PROGRAM MainState
VAR
	iMainSetp :INT;
	I1: UINT;
	iErrorSetp: INT;
	iLightSel: INT;
	bTurnOn: BOOL;
	bDoor_Stop: BOOL;
	I2: INT;
	I4: INT;
	I5: INT;
	i: UINT;
	iCode2: ICode;
	ExtSetVel: LREAL;
	ExtSetPos: LREAL;
	ExtSetAcc: LREAL;
	ExtSetDec: DINT;
	InitSetp: INT;
	rtStoping: R_TRIG;
	iMainInitSetp: INT;
	iMainEStopSetp: INT;
	K1: UINT;
	bInitReset: BOOL;
	DA1: INT;
	Code1: BOOL;
	Code2: BOOL;
	Code3: BOOL;
	Code4: BOOL;
	CyCtrl: INT;
	bWaterOn: BOOL;
	
	Execute: BOOL;
	bCoeWrite_GlueFeed: BOOL;
	bWaterOn2: BOOL;
	arrError:					ARRAY[1..10]OF BOOL;
	bEncloserEstop:BOOL;//外罩急停汇总
	bBoxEstop:BOOL;//按钮盒急停汇总
	F: INT;
	D195: MS_Alarm;
	D196: MS_Alarm;
	D197: MS_Alarm;
	D198: MS_Alarm;
	D199: MS_Alarm;
	D200: MS_Alarm;
	D201: MS_Alarm;
	D202: MS_Alarm;
	D203: MS_Alarm;
	D204: MS_Alarm;
	D205: MS_Alarm;
	D206: MS_Alarm;
	AnFD1: MS_Alarm;
	AnFD2: MS_Alarm;
	AnFD3: MS_Alarm;
	CaFD1: MS_Alarm;
	CaFD2: MS_Alarm;
	CaFD3: MS_Alarm;
	K2:INT;
	tCycleTimer: TON;
	bSave: BOOL;
	testii2: INT;
	bReadDataFirstCyle: BOOL;
	bReadDataCyle2: BOOL;
	bSaveTest: BOOL;
	rtSaveData: R_TRIG;
	CleanTrig: R_TRIG;
	CaCibang: R_TRIG;
	AnCibang: R_TRIG;
	CaCleanBrush:R_TRIG;
	AnCleanBrush:R_TRIG;
	
END_VAR

VAR
	R_TRIG_Bt: 			ARRAY[1..10]OF R_TRIG;
	TON20:Tc2_Standard.TON;	
//	TON21:Tc2_Standard.TON;	
	rt100:Tc2_Standard.R_TRIG;
	rt101:Tc2_Standard.R_TRIG;

	tDelayBuzze:TON;
	FanTon:TON;//除尘风机计时
	FanTonS:REAL;//除尘风机寿命秒
	FanTonH:REAL;//除尘风机寿命小时
	FanTonH_Set:REAL;//除尘风机寿命设定小时
	aAirAlarm_TON:TON;//气压报警延时；
	aTime:ARRAY[1..99] OF TON;//延时备用，1-16风速仪报警延时；
	aAlarm:ARRAY[1..99] OF BOOL;//报警预留;   1、气压不足报警；2、正极R角清废料报警；3、负极R角清废料报警；4、正极R角清废料计数错误；5、负极R角清废料计数错误；6、风机未启用报警；7、风机故障报警； 16-19、安全光栅报警；20-29、风速仪报警；30-47毛刷旋转感应报警，48毛刷旋转感应报警汇总,50:模切通道安全门报警；
	RT200:ARRAY[1..4] OF Tc2_Standard.R_TRIG;
	K3:INT;
	K4:INT;
	
	csAxis                 :ARRAY[1..MaxAxes] OF   CS_AxisCtrl;
	fbCy                   :ARRAY[1..MaxCy]    OF   FB_CylinderV2;
    fbRec                 :ARRAY[1..MaxRec]   OF   FB_Rectify;
	fbDustMotor       :ARRAY[1..MaxDust]   OF   CS_DustMoter;


    csCodeTcp:CS_CodeTcp;
    fbCamInTest: MC_CamIn;//主轴与驱动凸轮耦合

//速度模式验证
	MC_ExtSetPointGenDisable: MC_ExtSetPointGenDisable;
	MC_ExtSetPointGenEnable: MC_ExtSetPointGenEnable;
    MC_ExtSetPointGenOut:        Tc2_MC2.ST_McOutputs;
    MC_ExtSetPointGenOut2:        Tc2_MC2.ST_McOutputs;

    tonEStop:                     Tc2_Standard.TON;
   
  fbAnSetp1Moter  : CS_SetpMoter;
  fbCaSetp1Moter:CS_SetpMoter;
 // fbP4CutElectric_CY   :FB_Electric_CY;   电缸


	mc_Home    :MC_Home;

     fbCoeWrite_GlueFeed:       FB_EcCoeSdoWrite;
     	wEncodeHome                    :WORD:=6;
	test:ARRAY[1..10] OF BOOL;
	bAnReady:BOOL;//正极准备好
	bCaReady:BOOL;//负极准备好
	//fbDataXML       : FB_DataXML;
	rt10:Tc2_Standard.R_TRIG;
	testii:INT:=0;
	
	Code_MES				:ARRAY[1..20]OF  R_TRIG;
	fCode_MES				:ARRAY[1..20]OF  F_TRIG;
	tCode_MES				:ARRAY[1..20]OF  TON;
	
//模切直线电机COE寻址修改参数
	FB_EcCoESdoWrite_AnSEPTATCache : ARRAY[1..4] OF FB_EcCoESdoWrite; //正极极片缓存参数修改
	FB_EcCoESdoWrite_AnDriverDDR : ARRAY[1..4] OF FB_EcCoESdoWrite;	  //正极主驱参数修改
	FB_EcCoESdoWrite_CaSEPTATCache : ARRAY[1..4] OF FB_EcCoESdoWrite; //正极极片缓存参数修改
	FB_EcCoESdoWrite_CaDriverDDR : ARRAY[1..4] OF FB_EcCoESdoWrite;	  //正极主驱参数修改
	
	wSaveCoeCode  :DWORD:=16#65766173;    //电机参数保存
	
	SEPTATCache_fSmoothValue   :ARRAY[1..4] OF REAL;    //隔膜缓存写入参数值
	SEPTATCache_bWriteCoeValue  :ARRAY[1..4] OF BOOL;    //隔膜缓存写入执行	
	SEPTATCache_SavePara  :ARRAY[1..4] OF BOOL;   //隔膜缓存参数保存
	
	DriverDDR_fSmoothValue   :ARRAY[1..4] OF REAL;    //主驱写入参数值
	DriverDDR_bWriteCoeValue  :ARRAY[1..4] OF BOOL;    //主驱写入执行	
	DriverDDR_SavePara  :ARRAY[1..4] OF BOOL;   //主驱参数保存
	
	ExcelRate_R	:R_TRIG;	//Mes读取优报表	xfp20240316
	MTDWtStep: UINT;
	rDoorAlm :ARRAY[1..2]OF R_TRIG;
END_VAR

	aAirAlarm_TON(IN:=NOT I205[5],PT:=T#1S,Q=>);											
R_TRIG_Bt[1](CLK:= stSysState.btnStart OR stSysState.hmiStart);//启动上升沿
R_TRIG_Bt[2](CLK:= stSysState.btnStop  OR  stSysState.hmiStop);//停止上升沿
R_TRIG_Bt[4](CLK:=  stSysState.btnAuto OR  stSysState.hmiAuto);//手自动切换上升沿
R_TRIG_Bt[5](CLK:=  NOT stSysState.btnAuto);
R_TRIG_Bt[6](CLK:=stSysState.btnEstop);
R_TRIG_Bt[7](CLK:=stSysState.btnReset OR  stSysState.hmiReset );
R_TRIG_Bt[8](CLK:=  NOT stSysState.hmiAuto);



IF R_TRIG_Bt[4].Q THEN  //自动
	stSysState.FlgAuto:=TRUE;
	stSysState.FlgManua:=FALSE;
END_IF
IF R_TRIG_Bt[5].Q  OR  R_TRIG_Bt[8].Q   THEN  //手动
	stSysState.FlgAuto:=FALSE;
	stSysState.FlgManua:=TRUE;
	stSysState.bwindow:=FALSE;
END_IF
stSysState.bReset:=R_TRIG_Bt[7].Q  OR  bInitReset    ;  //复位

stSysState.bAnccdstate:= NOT AnAlarm.arrFlowAlarm[8] AND NOT AnAlarm.arrFlowAlarm[14] AND  ((NOT ProductPar.iModeEN.bCcdTcpEN AND NOT ProductPar.iModeEN.bSizeCCDEN  AND 
                         NOT  ProductPar.iModeEN.bChamferCCDEN AND NOT  ProductPar.iModeEN.bCuterCCDEN(* AND NOT  ProductPar.iModeEN.bLineScanCCDEN*)) OR  ProductPar.iModeEN.bP2PartEN);
stSysState.bCaccdstate:= NOT CaAlarm.arrFlowAlarm[8] AND NOT CaAlarm.arrFlowAlarm[14] AND  ((NOT ProductPar.iModeEN.bCcdTcpEN AND NOT ProductPar.iModeEN.bSizeCCDEN  AND 
                         NOT  ProductPar.iModeEN.bChamferCCDEN AND NOT  ProductPar.iModeEN.bCuterCCDEN (*AND NOT  ProductPar.iModeEN.bLineScanCCDEN*)) OR  ProductPar.iModeEN.bP2PartEN);

//////////////////////////////////系统流程///////////////////////
CASE iMainSetp OF 
0://   INIT
    Init();
    stSysState.iMode:=0;
 IF  stSysState.bInitDone THEN
     iMainSetp:=88;	
  END_IF
88://切换手动
  IF  stSysState.FlgManua THEN
	  iMainSetp:=300;
  END_IF
   
 (***********************手动*********************************) 
300:
   stSysState.iMode:=3;
   iMainSetp:=350;  
   
350: 
  	IF  R_TRIG_Bt[1].Q  AND stSysState.FlgAuto THEN  //启动按钮  
		IF stSysState.bAutoCondition THEN
		  stSysState.bwindow:=TRUE;	
	      iMainSetp:=90;
	    END_IF
	END_IF 
	
	IF  stSysState.FlgManua AND TON20.Q THEN  //系统清除
	   iMainSetp:=999;
	END_IF

 90:	
  	IF  R_TRIG_Bt[1].Q  AND stSysState.FlgAuto AND NOT stSysState.bwindow  THEN  //启动按钮  
		IF stSysState.bAutoCondition AND (stSysState.bAnccdstate OR ProductPar.iModeEN.iModeRun=1) AND (stSysState.bCaccdstate OR ProductPar.iModeEN.iModeRun=2) THEN
	      iMainSetp:=100;
	    END_IF
		
	ELSIF stSysState.FlgManua OR  stSysState.btnStop  OR  stSysState.hmiStop   OR   stSysState.bErrorStop OR 
          stSysState.btnEstop OR NOT stSysState.bAnccdstate OR NOT stSysState.bCaccdstate  THEN
		  iMainSetp:=300;
	END_IF 	
	
 (************************自动********************************) 
100:
   stSysState.iMode:=1;
   iMainSetp:=150;  
150:  //系统停止中......
    rtStoping(Clk:=stSysState.FlgManua OR  stSysState.btnStop  OR  stSysState.hmiStop   OR   stSysState.bErrorStop OR stSysState.btnEstop);  //自动中触发手动 停止 按钮  stSysRun.bErrorStop 包括正极和负极
    IF stSysState.FlgManua OR  stSysState.btnStop  OR  stSysState.hmiStop   OR   stSysState.bErrorStop OR stSysState.btnEstop THEN //自动触发停止 rtStoping.Q
		stSysState.Stoping:=TRUE;
		iMainSetp:=160; //
	END_IF;
	
160: //判断停止完成
   	IF  stSysState.bStopFinished  THEN
		AnSys.bStopFinished:=FALSE; 
		CaSys.bStopFinished:=FALSE;
       	stSysState.Stoping:=FALSE;
		IF NOT  stSysState.btnEstop THEN
			iMainSetp:=300; 
		ELSE
			stSysState.bInitDone:=FALSE;
			iMainSetp:=400; 	
		END_IF
	END_IF;
	
 (************************急停********************************) 
400://Stoping
   stSysState.iMode:=4;
    EStop();  
   iMainSetp:=450; 
      
450: //急停跳出 
	IF  NOT  stSysState.btnEstop  THEN  
        tonEStop(IN:=FALSE , PT:=T#50MS );
	    iMainSetp:=0;
    ELSE
         tonEStop(IN:=TRUE , PT:=T#50MS );
         IF  tonEStop.Q THEN
              tonEStop(IN:=FALSE , PT:=T#50MS );
              iMainSetp:=400;   
         END_IF
   	 END_IF

END_CASE


IF   stSysState.btnEstop   THEN  //AND  stSysState.iMode=3
	  iMainSetp:=400;
END_IF



(***************程序调用*********************)



AnPart(iMode:=stSysState.iMode);
CaPart(iMode:=stSysState.iMode);
//	XML();
   Condition();
    MotionBasic();
    CyBasic();
    RecBasic();
     Alarm();
     Pusle();
	 MS_Alarm();
	 Motion_coe();
	 MesCollect();
//PoleData.AnBeltData[1].Meney.SizeResults;

ACTION Alarm:

IF NOT ProductPar.iModeEN.bDoorEN THEN
	IF NOT I206[15] THEN
		aAlarm[49]:=TRUE;//模切通道安全门报警
	END_IF
END_IF



IF R_TRIG_Bt[7].Q THEN
	FOR K1:=1 TO MaxAxes DO 
     arrAxisAlarm[K1]:=  FALSE ;
END_FOR
END_IF
(******************气缸报警*******************)
FOR K1:=1 TO MaxCy DO 
     arrCYOnAlarm[K1]:=  arrCyCtrl[K1] .Status.Error1;
     arrCYOFFAlarm[K1]:=  arrCyCtrl[K1] .Status.Error2;
END_FOR
(******************正极气缸报警*******************)
bAnCYHaveAlarm:=FALSE;
FOR K1:=1 TO 20 DO 
      bAnCYHaveAlarm:=(bAnCYHaveAlarm OR arrCYOnAlarm[K1] OR  arrCYOFFAlarm[K1]) ;
END_FOR
FOR K1:=41 TO 60 DO 
      bAnCYHaveAlarm:=(bAnCYHaveAlarm OR arrCYOnAlarm[K1] OR  arrCYOFFAlarm[K1]) ;
END_FOR
(******************负极气缸报警*******************)
bCaCYHaveAlarm:=FALSE;
FOR K1:=21 TO 40 DO 
      bCaCYHaveAlarm:=(bCaCYHaveAlarm OR arrCYOnAlarm[K1] OR  arrCYOFFAlarm[K1]) ;
END_FOR
FOR K1:=61 TO MaxCy DO 
      bCaCYHaveAlarm:=(bCaCYHaveAlarm OR arrCYOnAlarm[K1] OR  arrCYOFFAlarm[K1]) ;
END_FOR

(******************切刀计数报警*************)
IF ProductPar.AnPar.iMouldCount1>= ProductPar.AnPar.iMouldCountAlarm1 THEN   //正极前模具切刀计数报警
	CuterCountAlarm[1]:=TRUE;
	ELSE
	CuterCountAlarm[1]:=FALSE;	
END_IF
(*IF ProductPar.AnPar.iMouldCount2>= ProductPar.AnPar.iMouldCountAlarm2 THEN   //正极后模具切刀计数报警
	CuterCountAlarm[2]:=TRUE;
	ELSE
	CuterCountAlarm[2]:=FALSE;	
END_IF*)
IF ProductPar.AnPar.iCuterCount>= ProductPar.AnPar.iCuterCountAlarm THEN   //正极裁切切刀计数报警
	CuterCountAlarm[3]:=TRUE;
	ELSE
	CuterCountAlarm[3]:=FALSE;	
END_IF
IF ProductPar.CaPar.iMouldCount1>= ProductPar.CaPar.iMouldCountAlarm1 THEN   //负极前模具切刀计数报警
	CuterCountAlarm[4]:=TRUE;
	ELSE
	CuterCountAlarm[4]:=FALSE;	
END_IF
(*IF ProductPar.CaPar.iMouldCount2>= ProductPar.CaPar.iMouldCountAlarm2 THEN   //负极后模具切刀计数报警
	CuterCountAlarm[5]:=TRUE;
	ELSE
	CuterCountAlarm[5]:=FALSE;	
END_IF*)
IF ProductPar.CaPar.iCuterCount>= ProductPar.CaPar.iCuterCountAlarm THEN   //负极裁切切刀计数报警
	CuterCountAlarm[6]:=TRUE;
	ELSE
	CuterCountAlarm[6]:=FALSE;	
END_IF

IF CuterCountAlarm[1] OR CuterCountAlarm[3] OR CuterCountAlarm[4] OR CuterCountAlarm[6] THEN// OR CuterCountAlarm[2] OR CuterCountAlarm[5]
	b_lifetime:=TRUE;
	ELSE
	b_lifetime:=FALSE;	
END_IF

IF ProductPar.AnPar.iCuterCount>= ProductPar.AnPar.iCuterCountWarning THEN    //正极裁切切刀计数预警
	CuterCountAlarm[7]:=TRUE;
	ELSE
	CuterCountAlarm[7]:=FALSE;	
END_IF
IF ProductPar.CaPar.iCuterCount>= ProductPar.CaPar.iCuterCountWarning THEN   //负极裁切切刀计数预警
	CuterCountAlarm[8]:=TRUE;
	ELSE
	CuterCountAlarm[8]:=FALSE;	
END_IF

(****************轴报警**************)
(*
FOR K1:=1 TO MaxAxes DO 
     arrAxisAlarm[K1]:=  arrAxis[K1] .Status.Error AND  arrAxis[K1] .Status.ErrorID<>16#42A0 OR NOT arrAxisCtrl[K1] .Status.Enabled ;
END_FOR
*)
(****************正极轴报警**************)
bAnAxisHaveAlarm:=FALSE;
FOR K1:=1 TO 15 DO 
		IF K1<>3 AND K1<>4 THEN
				arrAxisAlarm[K1]:=  arrAxis[K1] .Status.Error AND  arrAxis[K1] .Status.ErrorID<>16#42A0  ;//OR NOT arrAxisCtrl[K1] .Status.Enabled
				bAnAxisHaveAlarm:=bAnAxisHaveAlarm OR arrAxisAlarm[K1]  ;//OR arrAxisCtrl[K1] .Status.ErrorLimitSwitch
		END_IF
END_FOR

FOR K1:=18 TO 22 DO 
	  arrAxisAlarm[K1]:=  arrAxis[K1] .Status.Error AND  arrAxis[K1] .Status.ErrorID<>16#42A0  ;//OR NOT arrAxisCtrl[K1] .Status.Enabled
      bAnAxisHaveAlarm:=bAnAxisHaveAlarm OR arrAxisAlarm[K1]  ;//OR arrAxisCtrl[K1] .Status.ErrorLimitSwitch
END_FOR

FOR K1:=50 TO 52 DO 
	  arrAxisAlarm[K1]:=  arrAxis[K1] .Status.Error AND  arrAxis[K1] .Status.ErrorID<>16#42A0  ;//OR NOT arrAxisCtrl[K1] .Status.Enabled
      bAnAxisHaveAlarm:=bAnAxisHaveAlarm OR arrAxisAlarm[K1]  ;//OR arrAxisCtrl[K1] .Status.ErrorLimitSwitch
END_FOR

(****************负极轴报警**************)
bCaAxisHaveAlarm:=FALSE;
FOR K1:=25 TO 39 DO 
		IF K1<>27 AND K1<>28 THEN
				arrAxisAlarm[K1]:=  arrAxis[K1] .Status.Error AND  arrAxis[K1] .Status.ErrorID<>16#42A0  ;//OR NOT arrAxisCtrl[K1] .Status.Enabled
				bCaAxisHaveAlarm:=bCaAxisHaveAlarm OR arrAxisAlarm[K1]  ;//OR arrAxisCtrl[K1] .Status.ErrorLimitSwitch
		END_IF
END_FOR

FOR K1:=42 TO 46 DO 
	  arrAxisAlarm[K1]:=  arrAxis[K1] .Status.Error AND  arrAxis[K1] .Status.ErrorID<>16#42A0  ;//OR NOT arrAxisCtrl[K1] .Status.Enabled
      bCaAxisHaveAlarm:=bCaAxisHaveAlarm OR arrAxisAlarm[K1]  ;//OR arrAxisCtrl[K1] .Status.ErrorLimitSwitch
END_FOR

FOR K1:=56 TO 58 DO
	  arrAxisAlarm[K1]:=  arrAxis[K1] .Status.Error AND  arrAxis[K1] .Status.ErrorID<>16#42A0  ; //OR NOT arrAxisCtrl[K1] .Status.Enabled
      bCaAxisHaveAlarm:=bCaAxisHaveAlarm OR arrAxisAlarm[K1]  ;//OR arrAxisCtrl[K1] .Status.ErrorLimitSwitch
END_FOR

(******************张力报警*******************)
bAnTenHaveAlarm :=FALSE;
bCaTenHaveAlarm :=FALSE;
FOR K1:=1 TO 15 DO 
      bAnTenHaveAlarm:=bAnTenHaveAlarm OR AnAlarm.arrTenAlarm[K1];
	  bCaTenHaveAlarm:=bCaTenHaveAlarm OR CaAlarm.arrTenAlarm[K1];
END_FOR

(******************凸轮报警*******************)
bAnCreatTableHaveAlarm :=FALSE;
bCaCreatTableHaveAlarm :=FALSE;
bAnCamHaveAlarm :=FALSE;
bCaCamHaveAlarm :=FALSE;
FOR K1:=1 TO 30 DO 
      bAnCreatTableHaveAlarm:=bAnCreatTableHaveAlarm OR AnAlarm.arrCreatTableAlarm[K1];
	  bCaCreatTableHaveAlarm:=bCaCreatTableHaveAlarm OR CaAlarm.arrCreatTableAlarm[K1];
	  bAnCamHaveAlarm:=bAnCamHaveAlarm OR AnAlarm.arrCamInAlarm[K1];
	  bCaCamHaveAlarm:=bAnCamHaveAlarm OR CaAlarm.arrCamInAlarm[K1];
END_FOR

(******************齿轮报警*******************)
bAnGearHaveAlarm :=FALSE;
bCaGearHaveAlarm :=FALSE;
FOR K1:=1 TO 25 DO 
      bAnGearHaveAlarm:=bAnGearHaveAlarm OR AnAlarm.arrGearAlarm[K1];
	  bCaGearHaveAlarm:=bCaGearHaveAlarm OR CaAlarm.arrGearAlarm[K1];
END_FOR

(******************流程报警*******************)
bAnFlowHaveAlarm :=FALSE;
bCaFlowHaveAlarm :=FALSE;
FOR K1:=1 TO 50 DO 
      bAnFlowHaveAlarm:=bAnFlowHaveAlarm OR AnAlarm.arrFlowAlarm[K1];
	  bCaFlowHaveAlarm:=bCaFlowHaveAlarm OR CaAlarm.arrFlowAlarm[K1];
END_FOR

(******************提示*******************)
bAnHaveLightWarn :=FALSE;
bCaHaveLightWarn :=FALSE;
FOR K1:=1 TO 50 DO 
      bAnHaveLightWarn:=bAnHaveLightWarn OR AnAlarm.arrLightWarn[K1];
	  bCaHaveLightWarn:=bCaHaveLightWarn OR CaAlarm.arrLightWarn[K1];
END_FOR
(***DDR负数报警***)
(***DDR负数报警***)
IF arrAxisCtrl[NameNo.CaAxisNo.DriverDDR].Status.fActPos<-1 THEN
	CaAlarm.arrFlowAlarm[30]:=TRUE;
END_IF
IF arrAxisCtrl[NameNo.AnAxisNo.DriverDDR].Status.fActPos<-1 THEN
	AnAlarm.arrFlowAlarm[30]:=TRUE;
END_IF

 IF   stSysState.bReset AND  AnAlarm.arrFlowAlarm[30] THEN
	    arrAxisCtrl[NameNo.AnAxisNo.DriverDDR].Cmd.fSetPos:=360;
		arrAxisCtrl[NameNo.AnAxisNo.DriverDDR].Cmd.bSetPos:=TRUE;
		AnAlarm.arrFlowAlarm[30]:=FALSE;
ELSIF  stSysState.bReset AND CaAlarm.arrFlowAlarm[30] THEN
	    arrAxisCtrl[NameNo.CaAxisNo.DriverDDR].Cmd.fSetPos:=360;
		arrAxisCtrl[NameNo.CaAxisNo.DriverDDR].Cmd.bSetPos:=TRUE;
		CaAlarm.arrFlowAlarm[30]:=FALSE;
 END_IF

 (******************报警复位*****************)
 FOR K3:=1 TO 98 DO 
	IF   stSysState.bReset AND  aAlarm[K3]AND NOT aAlarm[52] AND NOT aAlarm[53] AND NOT aAlarm[54]  THEN
			aAlarm[K3]:=FALSE;
	END_IF
END_FOR

(***气压不足报警***)
IF aAirAlarm_TON.Q THEN
	aAlarm[1]:=TRUE;
END_IF
YL_Q[1]:=aAlarm[1];//气压报警传给叠台；
(*
(*** R角废料清洁提示***)
IF  YL_GVL2[1]>=YL_GVL2[2] THEN//正极R角清废料报警；
	aAlarm[2]:=TRUE;
END_IF

IF  YL_GVL2[1]< 0 THEN//正极R角清废料计数错误；
	aAlarm[4]:=TRUE;
END_IF
///////////////////////////
IF    YL_GVL2[3] >=YL_GVL2[4] THEN//负极R角清废料报警；
	aAlarm[3]:=TRUE;
END_IF

IF  YL_GVL2[3] < 0 THEN//负极R角清废料计数错误；
	aAlarm[5]:=TRUE;
END_IF
/////////////////////////////
//复位
IF   stSysState.bReset AND  (aAlarm[2] OR  aAlarm[4] )THEN
		YL_GVL2[1]:=0;
		aAlarm[2]:=FALSE;
		aAlarm[4]:=FALSE;
END_IF

IF   stSysState.bReset AND  (aAlarm[3] OR  aAlarm[5] )THEN
		YL_GVL2[3]:=0;
		aAlarm[3]:=FALSE;
		aAlarm[5]:=FALSE;
END_IF
*)
(*** 除尘风机报警提示***)
aAlarm[6];//风机未启用报警；
IF NOT ProductPar.iModeEN.bFounctionClose[2] THEN
		IF NOT YL_I[1] OR NOT YL_I[3] OR NOT YL_I[5] OR NOT YL_I[7] THEN//2个5.5KW的吸片风机,2个除尘风机；
			aAlarm[6]:=TRUE;//风机未启用报警；
		END_IF
		IF  YL_I[2] OR YL_I[4] OR YL_I[6] OR YL_I[8]  THEN
			aAlarm[7]:=TRUE;// 风机故障报警；
		END_IF
END_IF
FanTon(IN:=NOT aAlarm[6]AND NOT FanTon.Q,PT:=T#1S,Q=>);
IF FanTon.Q THEN
	FanTonS:=FanTonS+1;
END_IF
IF FanTonS>=3600 THEN
	FanTonH:=FanTonH+1;
	FanTonS:=0;
END_IF
IF FanTonH_Set>=FanTonH THEN
	aAlarm[61]:=TRUE;;//风机寿命报警
END_IF



(*** 除尘毛刷气缸没有升起报警***)

IF stSysState.iMode=1 AND NOT 	arrCyCtrl[NameNo.AnCYNo.PoleBrushDustPush_U].Io.DIOFFSwitch THEN
				aAlarm[8]:=TRUE;//	正极上表面毛刷除尘升降气缸位置异常；
END_IF
IF stSysState.iMode=1 AND NOT	arrCyCtrl[NameNo.AnCYNo.PoleWindDustPush_U].Io.DIOFFSwitch THEN
				aAlarm[9]:=TRUE;//	正极上表面风刀除尘升降气缸位置异常;
END_IF
IF stSysState.iMode=1 AND NOT	arrCyCtrl[NameNo.AnCYNo.PoleBrushDustPush_D].Io.DIOFFSwitch THEN
				aAlarm[10]:=TRUE;//	正极下表面毛刷除尘升降气缸位置异常;
END_IF
IF stSysState.iMode=1 AND NOT	arrCyCtrl[NameNo.AnCYNo.PoleWindDustPush_D].Io.DIOFFSwitch THEN
				aAlarm[11]:=TRUE;//	//	正极下表面风刀除尘升降气缸位置异常;
END_IF
////////////////////////
IF stSysState.iMode=1 AND NOT 	arrCyCtrl[NameNo.CaCYNo.PoleBrushDustPush_U].Io.DIOFFSwitch THEN
				aAlarm[12]:=TRUE;//	负极上表面毛刷除尘升降气缸位置异常；
END_IF
IF stSysState.iMode=1 AND NOT	arrCyCtrl[NameNo.CaCYNo.PoleWindDustPush_U].Io.DIOFFSwitch THEN
				aAlarm[13]:=TRUE;//	负极上表面风刀除尘升降气缸位置异常;
END_IF
IF stSysState.iMode=1 AND NOT	arrCyCtrl[NameNo.CaCYNo.PoleBrushDustPush_D].Io.DIOFFSwitch THEN
				aAlarm[14]:=TRUE;//	负极下表面毛刷除尘升降气缸位置异常;
END_IF
IF stSysState.iMode=1 AND NOT	arrCyCtrl[NameNo.CaCYNo.PoleWindDustPush_D].Io.DIOFFSwitch THEN
				aAlarm[15]:=TRUE;//	负极下表面风刀除尘升降气缸位置异常;
END_IF

(*** 安全光栅报警***)
IF NOT AnSenser.biSafetyCurtain_M THEN
	aAlarm[16]:=TRUE;
END_IF
IF NOT AnSenser.biSafetyCurtain_C THEN
	aAlarm[17]:=TRUE;
END_IF		
	
IF NOT CaSenser.biSafetyCurtain_M THEN
	aAlarm[18]:=TRUE;
END_IF
IF NOT CaSenser.biSafetyCurtain_C THEN
	aAlarm[19]:=TRUE;
END_IF	
	
(***************风速仪报警**************)
(***************风速仪报警**************)

aTime[1](IN:=I107[8],PT:=T#20S,Q=>	);
aTime[2](IN:=I107[9],PT:=T#20S,Q=>	);
aTime[3](IN:=I107[10],PT:=T#20S,Q=>	);
aTime[4](IN:=I107[11],PT:=T#20S,Q=>	);
aTime[5](IN:=I107[12],PT:=T#20S,Q=>	);

aTime[6](IN:=I207[8],PT:=T#20S,Q=>	);
aTime[7](IN:=I207[9],PT:=T#20S,Q=>	);
aTime[8](IN:=I207[10],PT:=T#20S,Q=>	);
aTime[9](IN:=I207[11],PT:=T#20S,Q=>	);
aTime[10](IN:=I207[12],PT:=T#20S,Q=>);

IF NOT ProductPar.iModeEN.bFounctionClose[1] THEN//风速仪屏蔽
	IF aTime[1].Q THEN
		aAlarm[20]:=TRUE;
	END_IF
	IF aTime[2].Q THEN
		aAlarm[21]:=TRUE;
	END_IF
	IF aTime[3].Q THEN
		aAlarm[22]:=TRUE;
	END_IF
	IF aTime[4].Q THEN
		aAlarm[23]:=TRUE;
	END_IF
	IF aTime[5].Q THEN
		aAlarm[24]:=TRUE;
	END_IF
	IF aTime[6].Q THEN
		aAlarm[25]:=TRUE;
	END_IF
	IF aTime[7].Q THEN
		aAlarm[26]:=TRUE;
	END_IF
	IF aTime[8].Q THEN
		aAlarm[27]:=TRUE;
	END_IF
	IF aTime[9].Q THEN
		aAlarm[28]:=TRUE;
	END_IF
	IF aTime[10].Q THEN
		aAlarm[29]:=TRUE;
	END_IF
ELSE
	FOR i:=20 TO 29 DO
		aAlarm[i]:=FALSE;
	END_FOR	
END_IF
(******************毛刷感应报警********************)
FOR K4:=30 TO 47 DO 
     aAlarm[48]:=  aAlarm[K4];
END_FOR
(*
(***********摆杆电机扭矩值设置过小报警************)
IF iTargetTorque[1]>-20 THEN
	aAlarm[50]:=TRUE;//正极；
END_IF
IF iTargetTorque[2]>-20 THEN
	aAlarm[51]:=TRUE;//负极；
END_IF
*)
(****************模切清洁报警*********************)

CleanTrig(CLK:= (ProductPar.CleanTimeHMIHour1 = System.StTime.wHour AND ProductPar.CleanTimeHMIMin1 =System.stTime.wMinute)
OR (ProductPar.CleanTimeHMIHour2 = System.StTime.wHour AND ProductPar.CleanTimeHMIMin2 =System.stTime.wMinute)
OR (ProductPar.CleanTimeHMIHour3 = System.StTime.wHour AND ProductPar.CleanTimeHMIMin3 =System.stTime.wMinute)
OR (ProductPar.CleanTimeHMIHour4 = System.StTime.wHour AND ProductPar.CleanTimeHMIMin4 =System.stTime.wMinute));
IF CleanTrig.Q THEN
	aAlarm[52]:=TRUE;//请清洁机台
END_IF
(****************磁棒校验时间报警******************)
AnCibang(CLK:= (ProductPar.CibangTimeHMIHour1 = System.StTime.wHour AND ProductPar.CibangTimeHMIDay1 =System.stTime.wDay));
CaCibang(CLK:= (ProductPar.CibangTimeHMIHour2 = System.StTime.wHour AND ProductPar.CibangTimeHMIDay2 =System.stTime.wDay));
IF AnCibang.Q THEN
	aAlarm[53]:=TRUE;//正极磁棒校验时间报警
END_IF
IF CaCibang.Q THEN
	aAlarm[54]:=TRUE;//负极磁棒校验时间报警
END_IF
(****************模切毛刷清洁时间****************)
AnCleanBrush(CLK:= (ProductPar.BrushTimeHMIHour1 = System.StTime.wHour AND ProductPar.BrushTimeHMIDay1 =System.stTime.wDay));
CaCleanBrush(CLK:= (ProductPar.BrushTimeHMIHour2 = System.StTime.wHour AND ProductPar.BrushTimeHMIDay2 =System.stTime.wDay));
IF AnCleanBrush.Q THEN
	aAlarm[62]:=TRUE;//正极毛刷清洁时间报警
END_IF
IF CaCleanBrush.Q THEN
	aAlarm[63]:=TRUE;//负极毛刷清洁时间报警
END_IF

IF NOT  DTM_Mes1.bFuncEN[0] AND NOT ProductPar.iModeEN.bP2PartEN AND (DTM_Mes1.bFuncEN[1] OR DTM_Mes1.bFuncEN[2] OR DTM_Mes1.bFuncEN[3] OR
	        DTM_Mes1.bFuncEN[4] OR DTM_Mes1.bFuncEN[5] OR DTM_Mes1.bFuncEN[6] OR DTM_Mes1.bFuncEN[7] )  THEN
		 aAlarm[64]:=TRUE;//模切有功能屏蔽报警
END_IF		
			


 AnAlarm.arrFlowAlarm[9];
AnAlarm.arrFlowAlarm[10];
AnAlarm.arrFlowAlarm[11];
AnAlarm.arrFlowAlarm[12];
AnAlarm.arrFlowAlarm[13];
CaAlarm.arrFlowAlarm[9];
CaAlarm.arrFlowAlarm[10];
CaAlarm.arrFlowAlarm[11];
CaAlarm.arrFlowAlarm[12];
CaAlarm.arrFlowAlarm[13];
(*===============================================报警信息============================================================*)
(*****************报警汇总****************)////根据实际情况汇总
//正极报警汇总
arrError[1]:=bAnAxisHaveAlarm OR bAnCYHaveAlarm OR bAnTenHaveAlarm OR bAnCreatTableHaveAlarm OR bAnCamHaveAlarm OR bAnGearHaveAlarm OR bAnFlowHaveAlarm OR aAlarm[16] OR aAlarm[17] OR aAlarm[49]
		OR AnAlarm.arrFlowAlarm[9] OR AnAlarm.arrFlowAlarm[10] OR AnAlarm.arrFlowAlarm[11] OR AnAlarm.arrFlowAlarm[12] OR AnAlarm.arrFlowAlarm[13]
		OR CaAlarm.arrFlowAlarm[9] OR CaAlarm.arrFlowAlarm[10] OR CaAlarm.arrFlowAlarm[11] OR CaAlarm.arrFlowAlarm[12] OR CaAlarm.arrFlowAlarm[13] OR CuterCountAlarm[3];
//负极报警汇总
arrError[2]:=bCaAxisHaveAlarm OR bCaCYHaveAlarm OR bCaTenHaveAlarm OR bCaCreatTableHaveAlarm OR bCaCamHaveAlarm OR bCaGearHaveAlarm OR bCaFlowHaveAlarm OR aAlarm[18] OR aAlarm[19] OR aAlarm[49]
		OR AnAlarm.arrFlowAlarm[9] OR AnAlarm.arrFlowAlarm[10] OR AnAlarm.arrFlowAlarm[11] OR AnAlarm.arrFlowAlarm[12] OR AnAlarm.arrFlowAlarm[13]
		OR CaAlarm.arrFlowAlarm[9] OR CaAlarm.arrFlowAlarm[10] OR CaAlarm.arrFlowAlarm[11] OR CaAlarm.arrFlowAlarm[12] OR CaAlarm.arrFlowAlarm[13] OR CuterCountAlarm[6];
//提示
arrError[3]:=(ProductPar.iModeEN.iModeRun=0 AND (bAnHaveLightWarn OR bCaHaveLightWarn)) OR
				   (ProductPar.iModeEN.iModeRun=1 AND bAnHaveLightWarn) OR 
				   (ProductPar.iModeEN.iModeRun=2 AND bCaHaveLightWarn);

arrError[4];
arrError[5]:=CaAlarm.arrFlowAlarm[30] OR AnAlarm.arrFlowAlarm[30] OR aAlarm[1] OR aAlarm[2] OR aAlarm[3] OR aAlarm[4] OR aAlarm[5]  OR aAlarm[6] OR aAlarm[7] OR aAlarm[8] OR aAlarm[9]
					OR aAlarm[10] OR aAlarm[11] OR aAlarm[12] OR aAlarm[13] OR aAlarm[14] OR aAlarm[15]OR aAlarm[52]OR aAlarm[53]OR aAlarm[54] ;

stSysState.bErrorStop:=(ProductPar.iModeEN.iModeRun=0 AND (arrError[1] OR arrError[2])) OR
								   (ProductPar.iModeEN.iModeRun=1 AND arrError[1]) OR 
								   (ProductPar.iModeEN.iModeRun=2 AND arrError[2])OR arrError[5] OR aAlarm[64];
								   
								   
rDoorAlm[1](CLK:=(AnAlarm.arrFlowAlarm[9] OR AnAlarm.arrFlowAlarm[10] OR AnAlarm.arrFlowAlarm[11] OR AnAlarm.arrFlowAlarm[12] OR AnAlarm.arrFlowAlarm[13]) AND NOT
                            bAnAxisHaveAlarm AND NOT bAnCYHaveAlarm AND NOT bAnTenHaveAlarm AND NOT bAnCreatTableHaveAlarm AND NOT bAnCamHaveAlarm AND NOT
                           bAnGearHaveAlarm AND NOT bAnFlowHaveAlarm AND NOT aAlarm[16] AND NOT aAlarm[17] AND NOT aAlarm[49]  AND NOT CuterCountAlarm[3] );
rDoorAlm[2](CLK:=(CaAlarm.arrFlowAlarm[9] OR CaAlarm.arrFlowAlarm[10] OR CaAlarm.arrFlowAlarm[11] OR CaAlarm.arrFlowAlarm[12] OR CaAlarm.arrFlowAlarm[13]) AND NOT 
                            bCaAxisHaveAlarm AND NOT bCaCYHaveAlarm AND NOT bCaTenHaveAlarm AND NOT bCaCreatTableHaveAlarm AND NOT bCaCamHaveAlarm AND NOT 
                            bCaGearHaveAlarm AND NOT bCaFlowHaveAlarm AND NOT aAlarm[18] AND NOT aAlarm[19] AND NOT aAlarm[49]AND NOT CuterCountAlarm[6] );
IF 	rDoorAlm[1].Q OR bCaDoorALM THEN						
	bAnDoorALM:=TRUE;
END_IF			

IF 	rDoorAlm[1].Q THEN						
	bCaDoorALM:=TRUE;
END_IF		

IF NOT stSysState.bErrorStop AND bAnDoorALM THEN
	bAnDoorALM:=FALSE;
END_IF		
	
IF NOT stSysState.bErrorStop AND bCaDoorALM THEN
	bCaDoorALM:=FALSE;
END_IF				
(*==============报警复位=========================*)
//轴  气缸报警  红灯亮       蜂鸣器 0.5秒 频率 响 8 秒后停止    

IF stSysState.iMode=3 THEN
	stSysState.bReset:=stSysState.btnReset;
END_IF

(*****蜂鸣器*****)
rt100(CLK:=stSysState.bErrorStop, Q=> );
rt101(CLK:=arrError[3]  , Q=> );
IF rt100.Q THEN
	iErrorSetp:=100;//故障报警
END_IF

IF rt101.Q THEN
	iErrorSetp:=200;//警告报警
END_IF


tDelayBuzze(IN:= , PT:= , Q=> , ET=> );
CASE iErrorSetp   OF
100:
  tDelayBuzze.PT:=T#8S;
  tDelayBuzze.IN:=TRUE;
  iErrorSetp:=500;
200:
  tDelayBuzze.PT:=T#4S;
   tDelayBuzze.IN:=TRUE;
  iErrorSetp:=600;
500:
		stSysState.boBuzzer:= Pulse._250ms.Q;  //   (NOT bError1 AND NOT bError2) AND
		IF tDelayBuzze.Q  THEN
			iErrorSetp:=0;
			tDelayBuzze.IN:=FALSE;
			stSysState.boBuzzer:=FALSE;
		END_IF
600:
	IF stSysState.iMode=1 AND NOT stSysState.bErrorStop THEN
		stSysState.boRedLight:=Pulse._1s.Q;
	END_IF
		stSysState.boBuzzer:= Pulse._1s.Q;  //    (NOT bError1 AND NOT bError2) AND
		IF tDelayBuzze.Q  THEN
			iErrorSetp:=0;
			tDelayBuzze.IN:=FALSE;
			IF stSysState.iMode=1 AND NOT stSysState.bErrorStop THEN
				stSysState.boRedLight:=FALSE;
			END_IF
			stSysState.boBuzzer:=FALSE;
		END_IF

END_CASE


(*****三色灯控制*********)
//自动   绿
    RT200[1](CLK:=stSysState.iMode=1 AND NOT stSysState.bErrorStop , Q=> ); 
   IF RT200[1].Q THEN
	  bTurnOn:=TRUE;
      iLightSel:=3;
   END_IF       
//手动  黄
    RT200[2](CLK:=stSysState.iMode=3 AND NOT stSysState.bErrorStop , Q=> ); 
   IF RT200[2].Q THEN
	  bTurnOn:=TRUE;
      iLightSel:=2;
   END_IF 

//暂停   黄
    RT200[3](CLK:=stSysState.iMode=2 AND NOT stSysState.bErrorStop , Q=> ); 
   IF RT200[3].Q THEN
	  bTurnOn:=TRUE;
      iLightSel:=2;
   END_IF 
   
//暂停   红   //急停 OR 故障
    RT200[4](CLK:=stSysState.iMode=4  OR stSysState.bErrorStop  , Q=> ); 
   IF RT200[4].Q THEN
	  bTurnOn:=TRUE;
      iLightSel:=1;
   END_IF    
   
IF bTurnOn THEN
	CASE iLightSel OF 
	  1: //红灯
		stSysState.boGreenLight:=FALSE;
		stSysState.boRedLight:=TRUE;
		stSysState.boYellowLight:=FALSE;
	
	  2://黄灯
		stSysState.boGreenLight:=FALSE;
		stSysState.boRedLight:=FALSE;
		stSysState.boYellowLight:=TRUE;
	
	  3://绿灯
		stSysState.boGreenLight:=TRUE;
		stSysState.boRedLight:=FALSE;
		stSysState.boYellowLight:=FALSE;
	
	END_CASE
   bTurnOn:=FALSE;
END_IF
arrAxis[4].Status.Homed;
arrAxis[5].Status.Homed;
arrAxis[6].Status.Homed;
arrAxis[7].Status.Homed;
arrAxis[8].Status.Homed;
arrAxis[9].Status.Homed;
arrAxis[10].Status.Homed;
arrAxis[11].Status.Homed;
arrAxis[12].Status.Homed;
arrAxis[13].Status.Homed;
arrAxis[14].Status.Homed;
arrAxis[15].Status.Homed;
arrAxis[16].Status.Homed;
arrAxis[17].Status.Homed;
arrAxis[18].Status.Homed;
arrAxis[19].Status.Homed;
arrAxis[20].Status.Homed;
arrAxis[21].Status.Homed;
arrAxis[22].Status.Homed;
arrAxis[23].Status.Homed;
arrAxis[24].Status.Homed;
arrAxis[25].Status.Homed;
arrAxis[26].Status.Homed;
arrAxis[27].Status.Homed;
arrAxis[28].Status.Homed;
arrAxis[29].Status.Homed;
arrAxis[30].Status.Homed;
arrAxis[31].Status.Homed;
arrAxis[32].Status.Homed;
arrAxis[33].Status.Homed;
arrAxis[34].Status.Homed;
arrAxis[35].Status.Homed;
arrAxis[36].Status.Homed;
arrAxis[37].Status.Homed;
arrAxis[38].Status.Homed;
arrAxis[39].Status.Homed;
arrAxis[40].Status.Homed;
arrAxis[41].Status.Homed;
arrAxis[42].Status.Homed;
arrAxis[43].Status.Homed;
arrAxis[44].Status.Homed;
arrAxis[45].Status.Homed;
arrAxis[46].Status.Homed;
arrAxis[47].Status.Homed;
arrAxis[48].Status.Homed;
arrAxis[49].Status.Homed;
arrAxis[50].Status.Homed;
arrAxis[51].Status.Homed;
arrAxis[52].Status.Homed;
arrAxis[53].Status.Homed;
arrAxis[54].Status.Homed;
arrAxis[55].Status.Homed;
arrAxis[56].Status.Homed;
arrAxis[57].Status.Homed;
arrAxis[58].Status.Homed;
arrAxis[59].Status.Homed;
arrAxis[60].Status.Homed;
END_ACTION

ACTION Condition:
//按钮汇总
stSysState.btnAuto:=AnSys.btnAuto AND CaSys.btnAuto ;
stSysState.btnStart:=AnSys.btnStart OR CaSys.btnStart;
stSysState.btnStop:=AnSys.btnStop OR CaSys.btnStop;
stSysState.btnReset:=AnSys.btnReset OR CaSys.btnReset;
bEncloserEstop:=(NOT AnBtn.EncloserEstop[1] OR NOT AnBtn.EncloserEstop[2] OR NOT AnBtn.EncloserEstop[3] OR 
						  NOT CaBtn.EncloserEstop[1] OR NOT CaBtn.EncloserEstop[2] OR NOT CaBtn.EncloserEstop[3])AND test[1] ;
bBoxEstop:=NOT AnBtn.PoleBoxEStop OR NOT AnBtn.NGBoxEStop OR  NOT CaBtn.PoleBoxEStop OR NOT CaBtn.NGBoxEStop ;

stSysState.btnEstop:=(NOT AnSys.btnEstop OR NOT CaSys.btnEstop //面板急停
								OR bEncloserEstop//外罩急停
								(*OR bBoxEstop//按钮盒急停*)
								) ;//常闭
//面板按钮灯控制
bAnReady:=AnSys.bAutoCondition1 AND AnSys.Homed AND NOT AnSys.hmiDisCamAll;
bCaReady:=CaSys.bAutoCondition1 AND CaSys.Homed AND NOT CaSys.hmiDisCamAll;

AnSys.boStartLight:=stSysState.boGreenLight OR bAnReady AND Pulse._500ms.Q OR AnSys.btnStart;
CaSys.boStartLight:=stSysState.boGreenLight OR bCaReady AND Pulse._500ms.Q OR AnSys.btnStart;

AnSys.boStopLight:=AnSys.Stoping AND Pulse._250ms.Q OR AnSys.btnStop;
CaSys.boStopLight:=CaSys.Stoping AND Pulse._250ms.Q OR CaSys.btnStop;

AnSys.boResetLight:=stSysState.boRedLight AND Pulse._500ms.Q OR AnSys.btnReset;
CaSys.boResetLight:=stSysState.boRedLight AND Pulse._500ms.Q OR CaSys.btnReset;		
////////////////////////////////////////////设备状态//////////////////////
	IF stSysState.btnEstop THEN
		stSysState.iModehmi:=4;
	ELSIF NOT stSysState.btnEstop AND stSysState.bErrorStop THEN
		stSysState.iModehmi:=5;
	ELSIF NOT stSysState.btnEstop AND NOT stSysState.bErrorStop AND stSysState.FlgManua AND stSysState.iMode=3THEN
		stSysState.iModehmi:=3;
	ELSIF NOT stSysState.btnEstop AND NOT stSysState.bErrorStop AND ((NOT stSysState.FlgManua AND stSysState.FlgAuto AND stSysState.iMode=1) OR stSysState.iMode=1) THEN
		stSysState.iModehmi:=1;
	ELSIF NOT stSysState.btnEstop AND NOT stSysState.bErrorStop AND NOT stSysState.FlgManua AND stSysState.FlgAuto AND stSysState.iMode<>1 AND
		 	((ProductPar.iModeEN.iModeRun=0 AND bAnReady AND bCaReady) OR (ProductPar.iModeEN.iModeRun=1 AND bAnReady) OR (ProductPar.iModeEN.iModeRun=2 AND bCaReady))
			THEN	
		stSysState.iModehmi:=2;	
	ELSE
		stSysState.iModehmi:=6;	
	END_IF		
	P2Interaction.bP1Runing:=stSysState.iModehmi=1;
////////////////////////////////////////////主流程与分模块交互//////////////////////
(*
stSysState.bAutoCondition:=((AnSys.bAutoCondition1 AND AnSys.Homed AND NOT AnSys.hmiDisCamAll AND 
			CaSys.bAutoCondition1 AND CaSys.Homed AND NOT CaSys.hmiDisCamAll AND
			ProductPar.iModeEN.iModeRun=0) OR//正负同时启用
			(AnSys.bAutoCondition1 AND AnSys.Homed AND NOT AnSys.hmiDisCamAll AND
			ProductPar.iModeEN.iModeRun=1) OR//仅正极启用
			(CaSys.bAutoCondition1 AND CaSys.Homed AND NOT CaSys.hmiDisCamAll AND
			ProductPar.iModeEN.iModeRun=2))//仅负极启用
			AND NOT stSysState.bErrorStop;
*)
stSysState.bAutoCondition:=	(AnSys.bAutoCondition1 AND AnSys.Homed AND NOT AnSys.hmiDisCamAll AND CaSys.bAutoCondition1 AND CaSys.Homed AND NOT CaSys.hmiDisCamAll AND ProductPar.iModeEN.iModeRun=0 
	AND	( (ProductPar.AnPar.MQ.bWindSelect AND  Ansys.PolePieceNumberOK1)  OR ( NOT ProductPar.AnPar.MQ.bWindSelect AND  Ansys.PolePieceNumberOK2) )
	AND  ( ( ProductPar.CaPar.MQ.bWindSelect AND  Casys.PolePieceNumberOK1 ) OR (  NOT ProductPar.CaPar.MQ.bWindSelect AND  Casys.PolePieceNumberOK2 ) ) ) OR //正负同时启用

		(AnSys.bAutoCondition1 AND AnSys.Homed AND NOT AnSys.hmiDisCamAll AND ProductPar.iModeEN.iModeRun=1  AND
		 ( ( ProductPar.AnPar.MQ.bWindSelect AND  Ansys.PolePieceNumberOK1 ) OR (  NOT ProductPar.AnPar.MQ.bWindSelect AND  Ansys.PolePieceNumberOK2 ) )) OR//仅正极启用
	
		(CaSys.bAutoCondition1 AND CaSys.Homed AND NOT CaSys.hmiDisCamAll AND ProductPar.iModeEN.iModeRun=2 AND 
		  ( ( ProductPar.CaPar.MQ.bWindSelect AND  Casys.PolePieceNumberOK1 ) OR (  NOT ProductPar.CaPar.MQ.bWindSelect AND  Casys.PolePieceNumberOK2 )  ) )//仅负极启用
		  AND NOT stSysState.bErrorStop; 			
Ansys.bAutoTen:=stSysState.iMode=1 AND (ProductPar.iModeEN.iModeRun=0 OR ProductPar.iModeEN.iModeRun=1);
Casys.bAutoTen:=stSysState.iMode=1 AND (ProductPar.iModeEN.iModeRun=0 OR ProductPar.iModeEN.iModeRun=2);
Ansys.bAutoMain:=AnSys.bAutoCondition2 AND ((ProductPar.iModeEN.iModeRun=0 AND CaSys.bAutoCondition2) OR ProductPar.iModeEN.iModeRun=1);
Casys.bAutoMain:=CaSys.bAutoCondition2 AND ((ProductPar.iModeEN.iModeRun=0 AND AnSys.bAutoCondition2) OR ProductPar.iModeEN.iModeRun=2);

stSysState.bStopFinished:=(AnSys.bStopFinished AND CaSys.bStopFinished  AND ProductPar.iModeEN.iModeRun=0) OR//正负同时启用
			(AnSys.bStopFinished AND ProductPar.iModeEN.iModeRun=1) OR//仅正极启用
			(CaSys.bStopFinished AND ProductPar.iModeEN.iModeRun=2);//仅负极启用

///////////////////////////////////交互映射/////////////////////////////////////
//////////叠片TO模切//////////
//一号叠台正极
AnInter.M1Done:=D_Pro.bAn_M1Done;
AnInter.M1Safety:=D_Pro.bAn_M1Safety;
AnInter.iM1Ask:=D_Sys.iAn1Ask;
AnInter.M1LockReady:=D_Pro.bAn_M1LockReady;
AnInter.M1JumpReady:=D_Pro.bAn_M1JumpReady;
AnInter.M1PoleHave:=D_Pro.bAn_M1PoleHave;


//一号叠台负极
CaInter.M1Done:=D_Pro.bCa_M1Done;
CaInter.M1Safety:=D_Pro.bCa_M1Safety;
CaInter.iM1Ask:=D_Sys.iCa1Ask;
CaInter.M1LockReady:=D_Pro.bCa_M1LockReady;
CaInter.M1JumpReady:=D_Pro.bCa_M1JumpReady;
CaInter.M1PoleHave:=D_Pro.bCa_M1PoleHave;


//二号叠台正极
AnInter.M2Done:=D_Pro.bAn_M2Done;
AnInter.M2Safety:=D_Pro.bAn_M2Safety;
AnInter.iM2Ask:=D_Sys.iAn2Ask;
AnInter.M2LockReady:=D_Pro.bAn_M2LockReady;
AnInter.M2JumpReady:=D_Pro.bAn_M2JumpReady;
AnInter.M2PoleHave:=D_Pro.bAn_M2PoleHave;


//二号叠台负极
CaInter.M2Done:=D_Pro.bCa_M2Done;
CaInter.M2Safety:=D_Pro.bCa_M2Safety;
CaInter.iM2Ask:=D_Sys.iCa2Ask;
CaInter.M2LockReady:=D_Pro.bCa_M2LockReady;
CaInter.M2JumpReady:=D_Pro.bCa_M2JumpReady;
CaInter.M2PoleHave:=D_Pro.bCa_M2PoleHave;


//三号叠台正极
AnInter.M3Done:=D_Pro.bAn_M3Done;
AnInter.M3Safety:=D_Pro.bAn_M3Safety;
AnInter.iM3Ask:=D_Sys.iAn3Ask;
AnInter.M3LockReady:=D_Pro.bAn_M3LockReady;
AnInter.M3JumpReady:=D_Pro.bAn_M3JumpReady;
AnInter.M3PoleHave:=D_Pro.bAn_M3PoleHave;


//三号叠台负极
CaInter.M3Done:=D_Pro.bCa_M3Done;
CaInter.M3Safety:=D_Pro.bCa_M3Safety;
CaInter.iM3Ask:=D_Sys.iCa3Ask;
CaInter.M3LockReady:=D_Pro.bCa_M3LockReady;
CaInter.M3JumpReady:=D_Pro.bCa_M3JumpReady;
CaInter.M3PoleHave:=D_Pro.bCa_M3PoleHave;


//公共
P2Interaction.bP2ClearDo:=D_Sys.bP2ClearDo;
P2Interaction.bP2ClearDone:=D_Sys.bP2ClearDone;
P2Interaction.P2M1Enable:=D_Sys.bP2M1Enable;//叠台工位：1=屏蔽   模切工位：1=启用，故取反。
P2Interaction.P2M2Enable:=D_Sys.bP2M2Enable;//叠台工位：1=屏蔽   模切工位：1=启用，故取反。
P2Interaction.P2M3Enable:=D_Sys.bP2M3Enable;//叠台工位：1=屏蔽   模切工位：1=启用，故取反。
P2Interaction.bP2Estop:=D_Sys.bP2Estop;
P2Interaction.bP2Runing:=D_Sys.bP2Runing;
P2Interaction.bP2Start:=D_Sys.bP2Start;

///////////模切TO叠片/////////
//一号叠台正极
M_Pro.bAn_M1Allow:=AnInter.M1Allow;
M_Pro.bAn_M1Allow2:=AnInter.M1Allow2;
//一号叠台负极
M_Pro.bCa_M1Allow:=CaInter.M1Allow;
//M_Pro.bCa_M1Allow:=CaInter.M1Allow2;
//二号叠台正极
M_Pro.bAn_M2Allow:=AnInter.M2Allow;
//M_Pro.bAn_M2Allow2:=AnInter.M2Allow2;
//二号叠台负极
M_Pro.bCa_M2Allow:=CaInter.M2Allow;
//M_Pro.bCa_M2Allow:=CaInter.M2Allow2;
//三号叠台正极
M_Pro.bAn_M3Allow:=AnInter.M3Allow;
//M_Pro.bAn_M3Allow2:=AnInter.M3Allow2;
//三号叠台负极
M_Pro.bCa_M3Allow:=CaInter.M3Allow;
//M_Pro.bCa_M3Allow:=CaInter.M3Allow2;

(*20240404
///////////模切TO叠片/////////
//一号叠台正极
M_Pro.bAn_M1Allow:=AnInter.M1Allow;
//一号叠台负极
M_Pro.bCa_M1Allow:=CaInter.M1Allow;
//二号叠台正极
M_Pro.bAn_M2Allow:=AnInter.M2Allow;
//二号叠台负极
M_Pro.bCa_M2Allow:=CaInter.M2Allow;
//三号叠台正极
M_Pro.bAn_M3Allow:=AnInter.M3Allow;
//三号叠台负极
M_Pro.bCa_M3Allow:=CaInter.M3Allow;
20240404*)
//公共
M_Sys.bP1ClearDo:=P2Interaction.bP1ClearDo;
M_Sys.bP1ClearDone:=P2Interaction.bP1ClearDone;
M_Sys.bP1Estop:=P2Interaction.bP1Estop;
M_Sys.bP1Runing:=P2Interaction.bP1Runing;
M_Sys.bP1Start:=P2Interaction.bP1Start;
M_Sys.iCarryPoleMode:=ProductPar.iModeEN.iCarryPoleMode;
M_Sys.p1state:=stSysState.iModehmi;
IF test[2] THEN
	MEMSET(ADR(PoleData.AnIntervalData),0,SIZEOF(PoleData.AnIntervalData)); //  
	test[2]:=FALSE;
END_IF
IF test[3] THEN
	MEMSET(ADR(PoleData.CaIntervalData),0,SIZEOF(PoleData.CaIntervalData)); //  
	test[3]:=FALSE;
END_IF
IF test[4] THEN
	MEMSET(ADR(PoleData.AnTabData),0,SIZEOF(PoleData.AnTabData)); //  
	test[4]:=FALSE;
END_IF
IF test[5] THEN
	MEMSET(ADR(PoleData.CaTabData),0,SIZEOF(PoleData.CaTabData)); //  
	test[5]:=FALSE;
END_IF
//监控
PoleData.	AnBeltData[1].bHavePole;
PoleData.	AnBeltData[2].bHavePole;
PoleData.	AnBeltData[3].bHavePole;
PoleData.	AnBeltData[4].bHavePole;
PoleData.	AnBeltData[5].bHavePole;
PoleData.	AnBeltData[6].bHavePole;
PoleData.	AnBeltData[7].bHavePole;
PoleData.	AnBeltData[8].bHavePole;
PoleData.	AnBeltData[9].bHavePole;
PoleData.	AnBeltData[10].bHavePole;
PoleData.	AnBeltData[11].bHavePole;
PoleData.	AnBeltData[12].bHavePole;
PoleData.	AnBeltData[13].bHavePole;
PoleData.	AnBeltData[14].bHavePole;
PoleData.	AnBeltData[15].bHavePole;
PoleData.	AnBeltData[16].bHavePole;
PoleData.	AnBeltData[17].bHavePole;
PoleData.	AnBeltData[18].bHavePole;
PoleData.	AnBeltData[19].bHavePole;
PoleData.	AnBeltData[20].bHavePole;
PoleData.	AnBeltData[21].bHavePole;
PoleData.	AnBeltData[22].bHavePole;
PoleData.	AnBeltData[23].bHavePole;
PoleData.	AnBeltData[24].bHavePole;
PoleData.	AnBeltData[25].bHavePole;
PoleData.	AnBeltData[26].bHavePole;
PoleData.	AnBeltData[27].bHavePole;
PoleData.	AnBeltData[28].bHavePole;
PoleData.	AnBeltData[29].bHavePole;
PoleData.	AnBeltData[30].bHavePole;				
stSysState.hmiStart;					
bInitReset;
arrAxisCtrl[NameNo.AnVirAxisNo.VirMain].Status.fModuloActPos;
arrAxisCtrl[NameNo.AnVirAxisNo.VirDriver].Status.fActPos;
arrAxisCtrl[NameNo.AnVirAxisNo.VirBelt].Status.fActPos;
arrAxisCtrl[NameNo.AnAxisNo.Mould].Status.fModuloActPos;
arrAxisCtrl[NameNo.AnAxisNo.Cuter].Status.fModuloActPos;
arrAxisCtrl[NameNo.AnAxisNo.DriverDDR].Status.fActPos;
arrAxisCtrl[NameNo.AnAxisNo.CCDPressPush].Status.fModuloActPos;
//arrAxisCtrl[NameNo.AnAxisNo.NGPush2].Status.fModuloActPos;
arrAxisCtrl[NameNo.AnAxisNo.CuterBelt].Status.fActPos;
arrAxisCtrl[NameNo.AnAxisNo.NGPushReverseBelt].Status.fActPos;
arrAxisCtrl[NameNo.AnAxisNo.DedustBelt].Status.fActPos;
arrAxisCtrl[NameNo.AnAxisNo.DedustReverseBelt].Status.fActPos;
arrAxisCtrl[NameNo.AnAxisNo.SubBelt1].Status.fActPos;
arrAxisCtrl[NameNo.AnAxisNo.SubBelt2].Status.fActPos;
arrAxisCtrl[NameNo.AnAxisNo.SubBelt3].Status.fActPos;

arrAxisCtrl[NameNo.AnAxisNo.CuterBeltChange].Status.Homed;
arrAxisCtrl[NameNo.AnAxisNo.CuterBeltChange].cmd.bHome;

PoleData.	CaBeltData[1].bHavePole;
PoleData.	CaBeltData[2].bHavePole;
PoleData.	CaBeltData[3].bHavePole;
PoleData.	CaBeltData[4].bHavePole;
PoleData.	CaBeltData[5].bHavePole;
PoleData.	CaBeltData[6].bHavePole;
PoleData.	CaBeltData[7].bHavePole;
PoleData.	CaBeltData[8].bHavePole;
PoleData.	CaBeltData[9].bHavePole;
PoleData.	CaBeltData[10].bHavePole;
PoleData.	CaBeltData[11].bHavePole;
PoleData.	CaBeltData[12].bHavePole;
PoleData.	CaBeltData[13].bHavePole;
PoleData.	CaBeltData[14].bHavePole;
PoleData.	CaBeltData[15].bHavePole;
PoleData.	CaBeltData[16].bHavePole;
PoleData.	CaBeltData[17].bHavePole;
PoleData.	CaBeltData[18].bHavePole;
PoleData.	CaBeltData[19].bHavePole;
PoleData.	CaBeltData[20].bHavePole;
PoleData.	CaBeltData[21].bHavePole;
PoleData.	CaBeltData[22].bHavePole;
PoleData.	CaBeltData[23].bHavePole;
PoleData.	CaBeltData[24].bHavePole;
PoleData.	CaBeltData[25].bHavePole;
PoleData.	CaBeltData[26].bHavePole;
PoleData.	CaBeltData[27].bHavePole;
PoleData.	CaBeltData[28].bHavePole;
PoleData.	CaBeltData[29].bHavePole;
PoleData.	CaBeltData[30].bHavePole;	




//正极左卷料号OK
IF  (ProductPar.AnPar.MQ.bWindSelect AND arrCyCtrl[NameNo.AnCYNo.Inflation_L].Status.ONState 
 AND DT_To_MQ_MES.Mes_PcToPlc1 AND  LEN(DT_To_MQ_MES.PostiveCode1)>6  )  OR ProductPar.iModeEN.PartNumberOff THEN
	Ansys.PolePieceNumberOK1:=TRUE;
ELSE
	Ansys.PolePieceNumberOK1:=FALSE;
END_IF

//正极右卷料号OK
IF  (NOT ProductPar.AnPar.MQ.bWindSelect AND arrCyCtrl[NameNo.AnCYNo.Inflation_R].Status.ONState
  AND DT_To_MQ_MES.Mes_PcToPlc2 AND LEN(DT_To_MQ_MES.PostiveCode2)>6  )  OR ProductPar.iModeEN.PartNumberOff THEN
	Ansys.PolePieceNumberOK2:=TRUE;
ELSE
	Ansys.PolePieceNumberOK2:=FALSE;
END_IF

//当前使用左卷
IF ProductPar.AnPar.MQ.bWindSelect THEN
	IF Ansys.PolePieceNumberOK1 THEN
		PoleData.AnBeltData[1].Code:=DT_To_MQ_MES.PostiveCode1;
	ELSE
		PoleData.AnBeltData[1].Code:='';//当前卷物料码异常
	END_IF
ELSE//当前使用右卷
	IF Ansys.PolePieceNumberOK2 THEN
		PoleData.AnBeltData[1].Code:=DT_To_MQ_MES.PostiveCode2;
	ELSE
		PoleData.AnBeltData[1].Code:='';//当前卷物料码异常
	END_IF
END_IF

//正极右卷换左卷---正常换卷
Code_MES[1](CLK:=ProductPar.AnPar.MQ.bWindSelect , Q=> );//AND arrCyCtrl[NameNo.AnCYNo.Inflation_L].Status.ONState  AND  stAnUwindTen.bTensionOK 
IF Code_MES[1].Q THEN
	Ansys.PolePieceNumberOK2:=FALSE;//正极右卷料号OK
	MQ_To_DT_MES.Mes_PlcToPc1:=FALSE;//正极左卷换卷请求
	MQ_To_DT_MES.Mes_PlcToPc2:=TRUE;//正极右卷换卷请求触发
END_IF
//正极左卷换右卷---正常换卷
Code_MES[2](CLK:=NOT ProductPar.AnPar.MQ.bWindSelect  , Q=> );//AND arrCyCtrl[NameNo.AnCYNo.Inflation_R].Status.ONState  AND  stAnUwindTen.bTensionOK
IF Code_MES[2].Q THEN
	Ansys.PolePieceNumberOK1:=FALSE;//正极左卷料号OK
	MQ_To_DT_MES.Mes_PlcToPc1:=TRUE;//正极左卷换卷请求触发
	MQ_To_DT_MES.Mes_PlcToPc2:=FALSE;//正极右卷换卷请求
END_IF

//正极气涨轴切换换卷
Code_MES[3](CLK:=arrCyCtrl[NameNo.AnCYNo.Inflation_L].Io.DOStatus1, Q=> );//左卷
Code_MES[4](CLK:=arrCyCtrl[NameNo.AnCYNo.Inflation_R].Io.DOStatus1, Q=> );//右卷
IF Code_MES[3].Q THEN//左卷请求
	Ansys.PolePieceNumberOK1:=FALSE;//正极左卷料号OK
	MQ_To_DT_MES.Mes_PlcToPc1:=TRUE;//正极左卷换卷请求触发
	MQ_To_DT_MES.Mes_PlcToPc2:=FALSE;//正极右卷换卷请求
END_IF
IF Code_MES[4].Q THEN//右卷请求
	Ansys.PolePieceNumberOK2:=FALSE;//正极右卷料号OK
	MQ_To_DT_MES.Mes_PlcToPc1:=FALSE;//正极左卷换卷请求
	MQ_To_DT_MES.Mes_PlcToPc2:=TRUE;//正极右卷换卷请求触发
END_IF



//负极左卷料号OK
IF  (ProductPar.CaPar.MQ.bWindSelect AND arrCyCtrl[NameNo.CaCYNo.Inflation_L].Status.ONState 
 AND DT_To_MQ_MES.Mes_PcToPlc3 AND  LEN(DT_To_MQ_MES.NegativeCode1)>6  )  OR ProductPar.iModeEN.PartNumberOff THEN
	Casys.PolePieceNumberOK1:=TRUE;
ELSE
	Casys.PolePieceNumberOK1:=FALSE;
END_IF

//负极右卷料号OK
IF  (NOT ProductPar.CaPar.MQ.bWindSelect AND arrCyCtrl[NameNo.CaCYNo.Inflation_R].Status.ONState
  AND DT_To_MQ_MES.Mes_PcToPlc4 AND LEN(DT_To_MQ_MES.NegativeCode2)>6  )  OR ProductPar.iModeEN.PartNumberOff THEN
	Casys.PolePieceNumberOK2:=TRUE;
ELSE
	Casys.PolePieceNumberOK2:=FALSE;
END_IF

IF ProductPar.CaPar.MQ.bWindSelect THEN
	IF  Casys.PolePieceNumberOK1 THEN
		PoleData.CaBeltData[1].Code:=DT_To_MQ_MES.NegativeCode1;
	ELSE
		PoleData.CaBeltData[1].Code:='';//当前卷物料码异常
	END_IF
ELSE
	IF  Casys.PolePieceNumberOK2 THEN
		PoleData.CaBeltData[1].Code:=DT_To_MQ_MES.NegativeCode2;
	ELSE
		PoleData.CaBeltData[1].Code:='';//当前卷物料码异常
	END_IF
END_IF

//负极右卷换左卷---正常换卷
Code_MES[5](CLK:=ProductPar.CaPar.MQ.bWindSelect  , Q=> );//AND arrCyCtrl[NameNo.CaCYNo.Inflation_L].Status.ONState  AND  stCaUwindTen.bTensionOK
IF Code_MES[5].Q THEN
	Casys.PolePieceNumberOK2:=FALSE;//负极右卷料号OK
	MQ_To_DT_MES.Mes_PlcToPc3:=FALSE;//负极左卷换卷请求
	MQ_To_DT_MES.Mes_PlcToPc4:=TRUE;//负极右卷换卷请求触发
END_IF
//正极左卷换右卷---正常换卷
Code_MES[6](CLK:=NOT ProductPar.CaPar.MQ.bWindSelect  , Q=> );//AND arrCyCtrl[NameNo.CaCYNo.Inflation_R].Status.ONState  AND  stCaUwindTen.bTensionOK
IF Code_MES[6].Q THEN
	Casys.PolePieceNumberOK1:=FALSE;//负极左卷料号OK
	MQ_To_DT_MES.Mes_PlcToPc3:=TRUE;//负极左卷换卷请求触发
	MQ_To_DT_MES.Mes_PlcToPc4:=FALSE;//负极右卷换卷请求
END_IF


//负极气涨轴切换换卷
Code_MES[7](CLK:=arrCyCtrl[NameNo.CaCYNo.Inflation_L].Io.DOStatus1, Q=> );//左卷
Code_MES[8](CLK:=arrCyCtrl[NameNo.CaCYNo.Inflation_R].Io.DOStatus1, Q=> );//右卷
IF Code_MES[7].Q THEN//左卷请求
	Casys.PolePieceNumberOK1:=FALSE;//负极左卷料号OK
	MQ_To_DT_MES.Mes_PlcToPc3:=TRUE;//负极左卷换卷请求触发
	MQ_To_DT_MES.Mes_PlcToPc4:=FALSE;//负极右卷换卷请求
END_IF
IF Code_MES[8].Q THEN//右卷请求
	Casys.PolePieceNumberOK2:=FALSE;//负极右卷料号OK
	MQ_To_DT_MES.Mes_PlcToPc3:=FALSE;//负极左卷换卷请求
	MQ_To_DT_MES.Mes_PlcToPc4:=TRUE;//负极右卷换卷请求触发
END_IF



//条码校验未完成提示
IF ProductPar.AnPar.MQ.bWindSelect AND  NOT Ansys.PolePieceNumberOK1  AND NOT ProductPar.iModeEN.PartNumberOff THEN
	AnAlarm.arrLightWarn[41]:=TRUE;//正极左卷物料码校验未通过
ELSE
	AnAlarm.arrLightWarn[41]:=FALSE;//正极左卷物料码校验未通过
END_IF
IF NOT ProductPar.AnPar.MQ.bWindSelect AND NOT Ansys.PolePieceNumberOK2  AND NOT ProductPar.iModeEN.PartNumberOff THEN
	AnAlarm.arrLightWarn[42]:=TRUE;//正极右卷物料码校验未通过
ELSE
	AnAlarm.arrLightWarn[42]:=FALSE;//正极右卷物料码校验未通过
END_IF

IF ProductPar.CaPar.MQ.bWindSelect AND  NOT Casys.PolePieceNumberOK1  AND NOT ProductPar.iModeEN.PartNumberOff THEN
	CaAlarm.arrLightWarn[41]:=TRUE;//负极左卷物料码校验未通过
ELSE
	CaAlarm.arrLightWarn[41]:=FALSE;//负极左卷物料码校验未通过
END_IF
IF NOT  ProductPar.CaPar.MQ.bWindSelect AND NOT Casys.PolePieceNumberOK2  AND NOT ProductPar.iModeEN.PartNumberOff THEN
	CaAlarm.arrLightWarn[42]:=TRUE;//负极右卷物料码校验未通过
ELSE
	CaAlarm.arrLightWarn[42]:=FALSE;//负极右卷物料码校验未通过
END_IF


//触发信号清除
tCode_MES[1](IN:=MQ_To_DT_MES.Mes_PlcToPc1 , PT:=T#0.2S , Q=> , ET=> );
tCode_MES[2](IN:=MQ_To_DT_MES.Mes_PlcToPc2 , PT:=T#0.2S , Q=> , ET=> );
tCode_MES[3](IN:=MQ_To_DT_MES.Mes_PlcToPc3 , PT:=T#0.2S , Q=> , ET=> );
tCode_MES[4](IN:=MQ_To_DT_MES.Mes_PlcToPc4 , PT:=T#0.2S , Q=> , ET=> );
IF tCode_MES[1].Q THEN
	MQ_To_DT_MES.Mes_PlcToPc1:=FALSE;//正极左卷换卷请求触发
END_IF
IF tCode_MES[2].Q THEN
	MQ_To_DT_MES.Mes_PlcToPc2:=FALSE;//正极右卷换卷请求触发
END_IF
IF tCode_MES[3].Q THEN
	MQ_To_DT_MES.Mes_PlcToPc3:=FALSE;//负极左卷换卷请求触发
END_IF
IF tCode_MES[4].Q THEN
	MQ_To_DT_MES.Mes_PlcToPc4:=FALSE;//负极右卷换卷请求触发
END_IF


//料号相同检测
IF  NOT ProductPar.iModeEN.PartNumberOff  THEN
	IF DT_To_MQ_MES.PostiveCode1 =DT_To_MQ_MES.PostiveCode2 AND DT_To_MQ_MES.PostiveCode1<>''  THEN
		aAlarm[55]:=TRUE;;//正极左卷和正极右卷料号相同
	END_IF
	IF DT_To_MQ_MES.PostiveCode1 =DT_To_MQ_MES.NegativeCode1 AND DT_To_MQ_MES.PostiveCode1<>''  THEN
		aAlarm[56]:=TRUE;;//正极左卷和负极左卷料号相同
	END_IF
	IF DT_To_MQ_MES.PostiveCode1 =DT_To_MQ_MES.NegativeCode2 AND DT_To_MQ_MES.PostiveCode1<>''  THEN
		aAlarm[57]:=TRUE;;//正极左卷与负极右卷料号相同
	END_IF
	
	IF DT_To_MQ_MES.PostiveCode2 =DT_To_MQ_MES.NegativeCode1 AND DT_To_MQ_MES.PostiveCode2<>''  THEN
		aAlarm[58]:=TRUE;;//正极右卷和负极左卷料号相同
	END_IF
	IF DT_To_MQ_MES.PostiveCode2 =DT_To_MQ_MES.NegativeCode2 AND DT_To_MQ_MES.PostiveCode2<>'' THEN
		aAlarm[59]:=TRUE;;//正极右卷和负极右卷料号相同
	END_IF
	
	IF DT_To_MQ_MES.NegativeCode1= DT_To_MQ_MES.NegativeCode2 AND DT_To_MQ_MES.NegativeCode1<>'' THEN 
		aAlarm[60]:=TRUE;;//负极左卷和负极右卷料号相同
	END_IF
END_IF

IF YL_I[20] THEN//叠台一正极送片流水线安全点动条件 
		arrAxisCtrl[20].Cmd.JogN_Condition:=TRUE;
		arrAxisCtrl[20].Cmd.JogP_Condition:=TRUE;
ELSE
		arrAxisCtrl[20].Cmd.JogN_Condition:=FALSE;
		arrAxisCtrl[20].Cmd.JogP_Condition:=FALSE;	
END_IF
IF YL_I[21] THEN//叠台一负极送片流水线安全点动条件 
		arrAxisCtrl[44].Cmd.JogN_Condition:=TRUE;
		arrAxisCtrl[44].Cmd.JogP_Condition:=TRUE;
ELSE
		arrAxisCtrl[44].Cmd.JogN_Condition:=FALSE;
		arrAxisCtrl[44].Cmd.JogP_Condition:=FALSE;		
END_IF

IF YL_I[22] THEN//叠台二正极送片流水线安全点动条件 
		arrAxisCtrl[21].Cmd.JogN_Condition:=TRUE;
		arrAxisCtrl[21].Cmd.JogP_Condition:=TRUE;
ELSE
		arrAxisCtrl[21].Cmd.JogN_Condition:=FALSE;
		arrAxisCtrl[21].Cmd.JogP_Condition:=FALSE;	
END_IF
IF YL_I[23] THEN//叠台二负极送片流水线安全点动条件 
		arrAxisCtrl[45].Cmd.JogN_Condition:=TRUE;
		arrAxisCtrl[45].Cmd.JogP_Condition:=TRUE;
ELSE
		arrAxisCtrl[45].Cmd.JogN_Condition:=FALSE;
		arrAxisCtrl[45].Cmd.JogP_Condition:=FALSE;	
END_IF

IF YL_I[24] THEN//叠台三正极送片流水线安全点动条件 
		arrAxisCtrl[22].Cmd.JogN_Condition:=TRUE;
		arrAxisCtrl[22].Cmd.JogP_Condition:=TRUE;
ELSE
		arrAxisCtrl[22].Cmd.JogN_Condition:=FALSE;
		arrAxisCtrl[22].Cmd.JogP_Condition:=FALSE;	
END_IF
IF YL_I[25] THEN//叠台三负极送片流水线安全点动条件
		arrAxisCtrl[46].Cmd.JogN_Condition:=TRUE;
		arrAxisCtrl[46].Cmd.JogP_Condition:=TRUE;
ELSE
		arrAxisCtrl[46].Cmd.JogN_Condition:=FALSE;
		arrAxisCtrl[46].Cmd.JogP_Condition:=FALSE;	
END_IF
END_ACTION

ACTION CyBasic:

//气缸控制   刷新周期可以慢
FOR i:=1 TO MaxCy DO
    fbCy[i](bReset:=stSysState.bReset , CyCtrl:=arrCyCtrl[i] );
END_FOR
END_ACTION

ACTION EStop:
 FOR I1:=1 TO MaxAxes BY 1 DO
	arrAxisCtrl[I1].Cmd. bHome:=FALSE;
	arrAxisCtrl[I1].Cmd. bJog_Bw:=FALSE;	
	arrAxisCtrl[I1].Cmd. bJog_Fw:=FALSE;		
    arrAxisCtrl[I1].Cmd. bMoveAbs:=FALSE;		
    arrAxisCtrl[I1].Cmd. bMoveRel:=FALSE;	
    arrAxisCtrl[I1].Cmd. bMoveVelo:=FALSE;		
    arrAxisCtrl[I1].Cmd.bMoveModulo:=FALSE;	
    arrAxisCtrl[I1].Cmd. bSetPos:=FALSE;	    	
    arrAxisCtrl[I1].Cmd. iGoSetPos:=0;	  		
	arrAxisCtrl[NameNo.AnAxisNo.PoleTension].cmd.bEnable:=FALSE;
	arrAxisCtrl[NameNo.CaAxisNo.PoleTension].cmd.bEnable:=FALSE;
	arrAxisCtrl[I1].Cmd. bStop:=TRUE;		
  END_FOR;
 FOR I1:=1 TO MaxDust BY 1 DO
	arrDustMotor[I1].bRun_BW:=FALSE;
	arrDustMotor[I1].bRun_FW:=FALSE;	
  END_FOR
  
stAnUwindTen.bTenExecute:=FALSE;//正极放卷张力
stAnAuxDriverTen.bTenExecute:=FALSE;//正极张力辅助驱动			
		
stCaUwindTen.bTenExecute:=FALSE;//负极放卷张力						
stCaAuxDriverTen.bTenExecute:=FALSE;//负极张力辅助驱动
 



  stSysState.bInitDone:=FALSE;
  AnSys.bStopFinished:=FALSE; 
  CaSys.bStopFinished:=FALSE;
  stSysState.Stoping:=FALSE;
  AnSys.Homed:=FALSE;
  CaSys.Homed:=FALSE;


///////
	arrAxisCtrl[NameNo. AnVirAxisNo.VirMain].cmd.bEnable:=FALSE;
	arrAxisCtrl[NameNo. AnVirAxisNo.VirMain].cmd.bHalt:=FALSE;

	arrAxisCtrl[NameNo. CaVirAxisNo.VirMain].cmd.bEnable:=FALSE;
	arrAxisCtrl[NameNo. CaVirAxisNo.VirMain].cmd.bHalt:=FALSE;
END_ACTION

ACTION Init:

//整机初始化
//所有轴上使能，凸轮创建，时间轴跑速度

CASE iMainInitSetp OF
0:
    IF  NOT   stSysState.bInitDone THEN
         iMainInitSetp:=10;
    END_IF
10:
    FOR i:=1 TO MaxAxes DO 
		arrAxisCtrl[i].Cmd.bEnable:=TRUE;
		arrAxisCtrl[i].Cmd.bEnableFw:=TRUE;
		arrAxisCtrl[i].Cmd.bEnableBw:=TRUE;
	(*其他操作指令*)  
		arrAxisCtrl[i].Cmd.bHome:=FALSE;
		arrAxisCtrl[i].Cmd.bJog_Bw:=FALSE;
		arrAxisCtrl[i].Cmd.bHalt:=FALSE;
		arrAxisCtrl[i].Cmd.bJog_Fw:=FALSE;
		arrAxisCtrl[i].Cmd.bMoveAbs:=FALSE;
		arrAxisCtrl[i].Cmd.bMoveVelo:=FALSE;
		arrAxisCtrl[i].Cmd.bMoveRel:=FALSE;
		arrAxisCtrl[i].Cmd.bReset:=FALSE;
		arrAxisCtrl[i].Cmd.bStop:=FALSE;
		arrAxisCtrl[i].Cmd.bSetPos:=FALSE;
		
		//arrAxisCtrl[i].Cmd.JogN_Condition:=TRUE;
		//arrAxisCtrl[i].Cmd.JogP_Condition:=TRUE;
		arrAxisCtrl[i].Cmd.Home_Condition:=TRUE;
		
		
    END_FOR
    K1:=0;
    iMainInitSetp:=20;
20: //复位一次
   bInitReset:=TRUE;
   iMainInitSetp:=30;
30:
   K1:=K1+1;
   IF  K1>=10 THEN
        bInitReset:=FALSE;
        iMainInitSetp:=40;
   ELSE
     iMainInitSetp:=20;
   END_IF

40://正负极 Init
   AnSys.bInit:=TRUE;
   CaSys.bInit:=TRUE;
   AnSys.bInitDone:=FALSE;
   CaSys.bInitDone:=FALSE;
   iMainInitSetp:=50;
50:
   IF  AnSys.bInitDone AND CaSys.bInitDone THEN //  
        iMainInitSetp:=60;
	   // AnSys.bInitDone:=FALSE;
	   // CaSys.bInitDone:=FALSE;		
    END_IF

60: //复位一次
   bInitReset:=TRUE;
   iMainInitSetp:=70;
   
70: //Time 轴跑速度
  IF  arrAxis[NameNo.VirTimeWind].Status.ControlLoopClosed THEN
	  arrAxisPar[NameNo.VirTimeWind].fVelocity_of_Velo:=100;
	  arrAxisCtrl[NameNo.VirTimeWind].Cmd.bMoveVelo:=TRUE;
      bInitReset:=FALSE;
	  iMainInitSetp:=80;
  END_IF
 
80:
  IF arrAxis[NameNo.VirTimeWind].Status.ConstantVelocity THEN
        stSysState.bInitDone:=TRUE;
        iMainInitSetp:=0;
  END_IF

END_CASE
END_ACTION

ACTION MesCollect:
//xfp20240315 与MES交互优报表
ExcelRate_R(clk:=(DTM_Mes1.uOther[0]=1),Q=>);	//MES读取触发上升沿
IF ExcelRate_R.Q THEN	
	MTDWtStep:=10;
END_IF	

CASE MTDWtStep OF
	10:
		IF system.stTime.wHour >=8 AND system.stTime.wHour <20 THEN
			MTD_Mes1.rExcelRate[0]:=An_Production.NgPerHourDayCount[49];//正极极片尺寸NG总数量
			MTD_Mes1.rExcelRate[1]:=An_Production.NgPerHourDayCount[1];//正极极片长度不良
			MTD_Mes1.rExcelRate[2]:=An_Production.NgPerHourDayCount[2];//正极极片CIL宽度不良
			MTD_Mes1.rExcelRate[3]:=An_Production.NgPerHourDayCount[3];//正极极片宽度不良
			MTD_Mes1.rExcelRate[4]:=An_Production.NgPerHourDayCount[4];//正极极耳宽度不良
			MTD_Mes1.rExcelRate[5]:=An_Production.NgPerHourDayCount[5];//正极极耳高度不良
			MTD_Mes1.rExcelRate[6]:=An_Production.NgPerHourDayCount[6];//正极极耳侧边距不良
			MTD_Mes1.rExcelRate[7]:=An_Production.NgPerHourDayCount[7];//正极极耳面积不良
			MTD_Mes1.rExcelRate[8]:=An_Production.NgPerHourDayCount[8];//正极圆角深度不良
			MTD_Mes1.rExcelRate[9]:=An_Production.NgPerHourDayCount[9];//极耳边缘角度不良
			MTD_Mes1.rExcelRate[10]:=An_Production.NgPerHourDayCount[10];//正极圆角宽度不良
			MTD_Mes1.rExcelRate[11]:=An_Production.NgPerHourDayCount[11];//正极圆角轮廓不良
			MTD_Mes1.rExcelRate[12]:=An_Production.NgPerHourDayCount[12];//正极圆角面积不良
			MTD_Mes1.rExcelRate[13]:=An_Production.NgPerHourDayCount[13];//正极圆角余料不良
			MTD_Mes1.rExcelRate[14]:=An_Production.NgPerHourDayCount[14];//正极尺寸其它不良
			MTD_Mes1.rExcelRate[15]:=An_Production.NgPerHourDayCount[48];//正极片线扫NG总数量
			MTD_Mes1.rExcelRate[16]:=An_Production.NgPerHourDayCount[21];//正极片抓边失败
			MTD_Mes1.rExcelRate[17]:=An_Production.NgPerHourDayCount[22];//正极片直边不良
			MTD_Mes1.rExcelRate[18]:=An_Production.NgPerHourDayCount[23];//正极片极片缺失
			MTD_Mes1.rExcelRate[19]:=An_Production.NgPerHourDayCount[24];//正极片接带
			MTD_Mes1.rExcelRate[20]:=An_Production.NgPerHourDayCount[26];//正极片漏金属
			MTD_Mes1.rExcelRate[21]:=An_Production.NgPerHourDayCount[27];//正极片气泡
			MTD_Mes1.rExcelRate[22]:=An_Production.NgPerHourDayCount[28];//正极片暗条纹
			MTD_Mes1.rExcelRate[23]:=An_Production.NgPerHourDayCount[29];//正极片亮条纹
			MTD_Mes1.rExcelRate[24]:=An_Production.NgPerHourDayCount[30];//正极片破损
			MTD_Mes1.rExcelRate[25]:=An_Production.NgPerHourDayCount[32];//通信超时
			MTD_Mes1.rExcelRate[26]:=An_Production.NgPerHourDayCount[34];//正极片其它NG
			MTD_Mes1.rExcelRate[27]:=Ca_Production.NgPerHourDayCount[49];//负极极片尺寸NG总数量
			MTD_Mes1.rExcelRate[28]:=Ca_Production.NgPerHourDayCount[1];//负极极片长度不良
			MTD_Mes1.rExcelRate[29]:=Ca_Production.NgPerHourDayCount[3];//负极极片宽度不良
			MTD_Mes1.rExcelRate[30]:=Ca_Production.NgPerHourDayCount[4];//负极极耳宽度不良
			MTD_Mes1.rExcelRate[31]:=Ca_Production.NgPerHourDayCount[5];//负极极耳高度不良
			MTD_Mes1.rExcelRate[32]:=Ca_Production.NgPerHourDayCount[6];//负极极耳边距不良
			MTD_Mes1.rExcelRate[33]:=Ca_Production.NgPerHourDayCount[7];//负极极耳面积不良
			MTD_Mes1.rExcelRate[34]:=Ca_Production.NgPerHourDayCount[8];//负极圆角深度不良
			MTD_Mes1.rExcelRate[35]:=Ca_Production.NgPerHourDayCount[9];//极耳边缘角度不良
			MTD_Mes1.rExcelRate[36]:=Ca_Production.NgPerHourDayCount[10];//负极圆角宽度不良
			MTD_Mes1.rExcelRate[37]:=Ca_Production.NgPerHourDayCount[11];//负极圆角轮廓不良
			MTD_Mes1.rExcelRate[38]:=Ca_Production.NgPerHourDayCount[12];//负极圆角面积不良
			MTD_Mes1.rExcelRate[39]:=Ca_Production.NgPerHourDayCount[13];//负极圆角余料不良
			MTD_Mes1.rExcelRate[40]:=Ca_Production.NgPerHourDayCount[14];//负极尺寸其它不良
			MTD_Mes1.rExcelRate[41]:=Ca_Production.NgPerHourDayCount[48];//负极片线扫NG总数量
			MTD_Mes1.rExcelRate[42]:=Ca_Production.NgPerHourDayCount[21];//负极片抓边失败
			MTD_Mes1.rExcelRate[43]:=Ca_Production.NgPerHourDayCount[22];//负极片直边不良
			MTD_Mes1.rExcelRate[44]:=Ca_Production.NgPerHourDayCount[23];//负极片极片缺失
			MTD_Mes1.rExcelRate[45]:=Ca_Production.NgPerHourDayCount[24];//负极片接带
			MTD_Mes1.rExcelRate[46]:=Ca_Production.NgPerHourDayCount[26];//负极片漏金属
			MTD_Mes1.rExcelRate[47]:=Ca_Production.NgPerHourDayCount[27];//负极片气泡
			MTD_Mes1.rExcelRate[48]:=Ca_Production.NgPerHourDayCount[28];//负极片暗条纹
			MTD_Mes1.rExcelRate[49]:=Ca_Production.NgPerHourDayCount[29];//负极片亮条纹
			MTD_Mes1.rExcelRate[50]:=Ca_Production.NgPerHourDayCount[30];//负极片破损
			MTD_Mes1.rExcelRate[51]:=Ca_Production.NgPerHourDayCount[32];//通信超时
			MTD_Mes1.rExcelRate[52]:=Ca_Production.NgPerHourDayCount[34];//	负极片其它NG
			MTD_Mes1.rExcelRate[53]:=An_Production.NgPerHourDayCount[25];//	正极线扫黄标
			MTD_Mes1.rExcelRate[54]:=An_Production.NgPerHourDayCount[31];//	正极线扫碎屑
			MTD_Mes1.rExcelRate[55]:=An_Production.NgPerHourDayCount[33];//	正极线扫脱碳
			MTD_Mes1.rExcelRate[56]:=Ca_Production.NgPerHourDayCount[25];//	负极线扫黄标
			MTD_Mes1.rExcelRate[57]:=Ca_Production.NgPerHourDayCount[31];//	负极线扫碎屑
			MTD_Mes1.rExcelRate[58]:=Ca_Production.NgPerHourDayCount[33];//	负极线扫脱碳
			MTD_Mes1.uOther[0]:=2;	//plc数据写入完成
			MTDWtStep:=20;
		ELSIF system.stTime.wHour >=20 OR system.stTime.wHour<8 THEN	
			MTD_Mes1.rExcelRate[0]:=An_Production.NgPerHourNightCount[49];//正极极片尺寸NG总数量
			MTD_Mes1.rExcelRate[1]:=An_Production.NgPerHourNightCount[1];//正极极片长度不良
			MTD_Mes1.rExcelRate[2]:=An_Production.NgPerHourNightCount[2];//正极极片CIL宽度不良
			MTD_Mes1.rExcelRate[3]:=An_Production.NgPerHourNightCount[3];//正极极片宽度不良
			MTD_Mes1.rExcelRate[4]:=An_Production.NgPerHourNightCount[4];//正极极耳宽度不良
			MTD_Mes1.rExcelRate[5]:=An_Production.NgPerHourNightCount[5];//正极极耳高度不良
			MTD_Mes1.rExcelRate[6]:=An_Production.NgPerHourNightCount[6];//正极极耳侧边距不良
			MTD_Mes1.rExcelRate[7]:=An_Production.NgPerHourNightCount[7];//正极极耳面积不良
			MTD_Mes1.rExcelRate[8]:=An_Production.NgPerHourNightCount[8];//正极圆角深度不良
			MTD_Mes1.rExcelRate[9]:=An_Production.NgPerHourNightCount[9];//极耳边缘角度不良
			MTD_Mes1.rExcelRate[10]:=An_Production.NgPerHourNightCount[10];//正极圆角宽度不良
			MTD_Mes1.rExcelRate[11]:=An_Production.NgPerHourNightCount[11];//正极圆角轮廓不良
			MTD_Mes1.rExcelRate[12]:=An_Production.NgPerHourNightCount[12];//正极圆角面积不良
			MTD_Mes1.rExcelRate[13]:=An_Production.NgPerHourNightCount[13];//正极圆角余料不良
			MTD_Mes1.rExcelRate[14]:=An_Production.NgPerHourNightCount[14];//正极尺寸其它不良
			MTD_Mes1.rExcelRate[15]:=An_Production.NgPerHourNightCount[48];//正极片线扫NG总数量
			MTD_Mes1.rExcelRate[16]:=An_Production.NgPerHourNightCount[21];//正极片抓边失败
			MTD_Mes1.rExcelRate[17]:=An_Production.NgPerHourNightCount[22];//正极片直边不良
			MTD_Mes1.rExcelRate[18]:=An_Production.NgPerHourNightCount[23];//正极片极片缺失
			MTD_Mes1.rExcelRate[19]:=An_Production.NgPerHourNightCount[24];//正极片接带
			MTD_Mes1.rExcelRate[20]:=An_Production.NgPerHourNightCount[26];//正极片漏金属
			MTD_Mes1.rExcelRate[21]:=An_Production.NgPerHourNightCount[27];//正极片气泡
			MTD_Mes1.rExcelRate[22]:=An_Production.NgPerHourNightCount[28];//正极片亮条纹
			MTD_Mes1.rExcelRate[23]:=An_Production.NgPerHourNightCount[29];//正极片亮条纹
			MTD_Mes1.rExcelRate[24]:=An_Production.NgPerHourNightCount[30];//正极片破损
			MTD_Mes1.rExcelRate[25]:=An_Production.NgPerHourNightCount[32];//通信超时
			MTD_Mes1.rExcelRate[26]:=An_Production.NgPerHourNightCount[34];//正极片其它NG
			MTD_Mes1.rExcelRate[27]:=Ca_Production.NgPerHourNightCount[49];//负极极片尺寸NG总数量
			MTD_Mes1.rExcelRate[28]:=Ca_Production.NgPerHourNightCount[1];//负极极片长度不良
			MTD_Mes1.rExcelRate[29]:=Ca_Production.NgPerHourNightCount[3];//负极极片宽度不良
			MTD_Mes1.rExcelRate[30]:=Ca_Production.NgPerHourNightCount[4];//负极极耳宽度不良
			MTD_Mes1.rExcelRate[31]:=Ca_Production.NgPerHourNightCount[5];//负极极耳高度不良
			MTD_Mes1.rExcelRate[32]:=Ca_Production.NgPerHourNightCount[6];//负极极耳边距不良
			MTD_Mes1.rExcelRate[33]:=Ca_Production.NgPerHourNightCount[7];//负极极耳面积不良
			MTD_Mes1.rExcelRate[34]:=Ca_Production.NgPerHourNightCount[8];//负极圆角深度不良
			MTD_Mes1.rExcelRate[35]:=Ca_Production.NgPerHourNightCount[9];//极耳边缘角度不良
			MTD_Mes1.rExcelRate[36]:=Ca_Production.NgPerHourNightCount[10];//负极圆角宽度不良
			MTD_Mes1.rExcelRate[37]:=Ca_Production.NgPerHourNightCount[11];//负极圆角轮廓不良
			MTD_Mes1.rExcelRate[38]:=Ca_Production.NgPerHourNightCount[12];//负极圆角面积不良
			MTD_Mes1.rExcelRate[39]:=Ca_Production.NgPerHourNightCount[13];//负极圆角余料不良
			MTD_Mes1.rExcelRate[40]:=Ca_Production.NgPerHourNightCount[14];//负极尺寸其它不良
			MTD_Mes1.rExcelRate[41]:=Ca_Production.NgPerHourNightCount[48];//负极片线扫NG总数量
			MTD_Mes1.rExcelRate[42]:=Ca_Production.NgPerHourNightCount[21];//负极片抓边失败
			MTD_Mes1.rExcelRate[43]:=Ca_Production.NgPerHourNightCount[22];//负极片直边不良
			MTD_Mes1.rExcelRate[44]:=Ca_Production.NgPerHourNightCount[23];//负极片极片缺失
			MTD_Mes1.rExcelRate[45]:=Ca_Production.NgPerHourNightCount[24];//负极片接带
			MTD_Mes1.rExcelRate[46]:=Ca_Production.NgPerHourNightCount[26];//负极片漏金属
			MTD_Mes1.rExcelRate[47]:=Ca_Production.NgPerHourNightCount[27];//负极片气泡
			MTD_Mes1.rExcelRate[48]:=Ca_Production.NgPerHourNightCount[28];//负极片暗条纹
			MTD_Mes1.rExcelRate[49]:=Ca_Production.NgPerHourNightCount[29];//负极片亮条纹
			MTD_Mes1.rExcelRate[50]:=Ca_Production.NgPerHourNightCount[30];//负极片破损
			MTD_Mes1.rExcelRate[51]:=Ca_Production.NgPerHourNightCount[32];//通信超时
			MTD_Mes1.rExcelRate[52]:=Ca_Production.NgPerHourNightCount[34];//负极片其它NG
			MTD_Mes1.rExcelRate[53]:=An_Production.NgPerHourNightCount[25];//	正极线扫黄标
			MTD_Mes1.rExcelRate[54]:=An_Production.NgPerHourNightCount[31];//	正极线扫碎屑	
			MTD_Mes1.rExcelRate[55]:=An_Production.NgPerHourNightCount[33];//	正极线扫脱碳
			MTD_Mes1.rExcelRate[56]:=Ca_Production.NgPerHourNightCount[25];//	负极线扫黄标	
			MTD_Mes1.rExcelRate[57]:=Ca_Production.NgPerHourNightCount[31];//	负极线扫碎屑
			MTD_Mes1.rExcelRate[58]:=Ca_Production.NgPerHourNightCount[33];//	负极线扫脱碳
			MTD_Mes1.uOther[0]:=2;	//plc数据写入完成
			MTDWtStep:=20;
		END_IF			
	20:
		IF DTM_Mes1.uOther[0]=0 THEN
			MTD_Mes1.uOther[0]:=0;
			MTDWtStep:=0;
		END_IF
END_CASE
(*
//功能开关状态
        MTD_Mes1.bFuncEN[1]:=ProductPar.iModeEN.bCcdTcpEN;
		MTD_Mes1.bFuncEN[2]:=ProductPar.iModeEN.bLineScanCCDEN;
	    MTD_Mes1.bFuncEN[3]:=ProductPar.iModeEN.bChamferCCDEN;		
	    MTD_Mes1.bFuncEN[4]:=ProductPar.iModeEN.bCuterCCDEN;		
	    MTD_Mes1.bFuncEN[5]:=ProductPar.iModeEN.bSizeCCDEN;	
        MTD_Mes1.bFuncEN[6]:=ProductPar.iModeEN.PartNumberOff;
		MTD_Mes1.bFuncEN[7]:=ProductPar.iModeEN.bTabWidtNGoff;*)
		
//模具切刀计数		
		MTD_Mes1.uOther[1]:=ProductPar.AnPar.iCuterCount;
		MTD_Mes1.uOther[2]:=ProductPar.CaPar.iCuterCount;
		MTD_Mes1.uOther[3]:=ProductPar.AnPar.iMouldCount1;
		MTD_Mes1.uOther[4]:=ProductPar.CaPar.iMouldCount1;		
	    MTD_Mes1.uOther[5]:=ProductPar.AnPar.iCuterCountAlarm;
		MTD_Mes1.uOther[6]:=ProductPar.CaPar.iCuterCountAlarm;
		MTD_Mes1.uOther[7]:=ProductPar.AnPar.iMouldCountAlarm1;
		MTD_Mes1.uOther[8]:=ProductPar.CaPar.iMouldCountAlarm1;
		MTD_Mes1.bFuncEN[8]:=ProductPar.AnPar.iCuterclear;
		MTD_Mes1.bFuncEN[9]:=ProductPar.CaPar.iCuterclear;
		MTD_Mes1.bFuncEN[10]:=ProductPar.AnPar.iMouldclear1;
		MTD_Mes1.bFuncEN[11]:=ProductPar.CaPar.iMouldclear1;
END_ACTION

ACTION Motion_coe:

//nSlaveAddr :ARRAY[1..6] OF INT :=[1003,1008,1018,1019,1020,1021] ;     //EtherCAT支路驱动器ID



//////////////////////////////////////////////////////////////////////正极////////////////////////////////////////////////////////////////
(*
//正极模切缓存
//写入
FB_EcCoESdoWrite_AnSEPTATCache[1](
	sNetId:= '192.168.10.10.4.1', 
	nSlaveAddr:=1025,   //模切缓存
	nSubIndex:=0 , 
	nIndex:=16#2108 ,   //  平滑时间
	pSrcBuf:=ADR(SEPTATCache_fSmoothValue[1]),       //写入参数值 
	cbBufLen:=SIZEOF(SEPTATCache_fSmoothValue[1]),    
	bExecute:= SEPTATCache_bWriteCoeValue[1],    
	tTimeout:= T#3S, 
	bBusy=> , 
	bError=> , 
	nErrId=> );
//保存	
FB_EcCoESdoWrite_AnSEPTATCache[3](
	sNetId:= '192.168.10.10.4.1', 
	nSlaveAddr:=1025 ,   //模切缓存
	nSubIndex:=0 , 
	nIndex:=16#2108 ,   // 平滑时间
	pSrcBuf:=ADR(wSaveCoeCode),      //保存参数值
	cbBufLen:=SIZEOF(wSaveCoeCode),    
	bExecute:=SEPTATCache_SavePara[1],    
	tTimeout:= T#3S, 
	bBusy=> , 
	bError=> , 
	nErrId=> );	
	
	
//写入	
FB_EcCoESdoWrite_AnSEPTATCache[2](
	sNetId:='192.168.10.10.4.1', 
	nSlaveAddr:=1025 ,   //模切缓存
	nSubIndex:=0 , 
	nIndex:=16#2109 ,   // 平滑方式
	pSrcBuf:=ADR(SEPTATCache_fSmoothValue[2]),       //写入参数值 
	cbBufLen:=SIZEOF(SEPTATCache_fSmoothValue[2]),    
	bExecute:=SEPTATCache_bWriteCoeValue[2],    
	tTimeout:= T#3S, 
	bBusy=> , 
	bError=> , 
	nErrId=> );	
//保存
FB_EcCoESdoWrite_AnSEPTATCache[4](
	sNetId:= '192.168.10.10.4.1', 
	nSlaveAddr:=1025,   //模切缓存
	nSubIndex:=0 , 
	nIndex:=16#2109 ,   // 平滑方式
	pSrcBuf:=ADR(wSaveCoeCode),      //保存参数值
	cbBufLen:=SIZEOF(wSaveCoeCode),    
	bExecute:=SEPTATCache_SavePara[2],    
	tTimeout:= T#3S, 
	bBusy=> , 
	bError=> , 
	nErrId=> );	


	
	
	
	
//正极模切主驱
//写入
FB_EcCoESdoWrite_AnDriverDDR[1](
	sNetId:= '192.168.10.10.4.1', 
	nSlaveAddr:=1026 ,   //模切主驱
	nSubIndex:=0 , 
	nIndex:=16#2108 ,   //  平滑时间
	pSrcBuf:=ADR(DriverDDR_fSmoothValue[1]),       //写入参数值 
	cbBufLen:=SIZEOF(DriverDDR_fSmoothValue[1]),    
	bExecute:= DriverDDR_bWriteCoeValue[1],    
	tTimeout:= T#3S, 
	bBusy=> , 
	bError=> , 
	nErrId=> );
//保存	
FB_EcCoESdoWrite_AnDriverDDR[3](
	sNetId:= '192.168.10.10.4.1', 
	nSlaveAddr:=1026 ,   //模切主驱
	nSubIndex:=0 , 
	nIndex:=16#2108 ,   // 平滑时间
	pSrcBuf:=ADR(wSaveCoeCode),      //保存参数值
	cbBufLen:=SIZEOF(wSaveCoeCode),    
	bExecute:= DriverDDR_SavePara[1],    
	tTimeout:= T#3S, 
	bBusy=> , 
	bError=> , 
	nErrId=> );	
	
	
	
	
//写入	
FB_EcCoESdoWrite_AnDriverDDR[2](
	sNetId:='192.168.10.10.4.1', 
	nSlaveAddr:=1026 ,   //模切主驱
	nSubIndex:=0 , 
	nIndex:=16#2109 ,   // 平滑方式
	pSrcBuf:=ADR(DriverDDR_fSmoothValue[2]), 
	cbBufLen:=SIZEOF(DriverDDR_fSmoothValue[2]),    
	bExecute:= DriverDDR_bWriteCoeValue[2],    
	tTimeout:= T#3S, 
	bBusy=> , 
	bError=> , 
	nErrId=> );	
//保存
FB_EcCoESdoWrite_AnDriverDDR[4](
	sNetId:= '192.168.10.10.4.1', 
	nSlaveAddr:=1026 ,   //模切主驱
	nSubIndex:=0 , 
	nIndex:=16#2109 ,   // 平滑方式
	pSrcBuf:=ADR(wSaveCoeCode),  
	cbBufLen:=SIZEOF(wSaveCoeCode),    
	bExecute:= DriverDDR_SavePara[2],    
	tTimeout:= T#3S, 
	bBusy=> , 
	bError=> , 
	nErrId=> );	
			
	



	
	
	
	
	
	
	
	
	
	

//////////////////////////////////////////////////////////////////////负极////////////////////////////////////////////////////////////////////

//负极模切缓存
//写入
FB_EcCoESdoWrite_CaSEPTATCache[1](
	sNetId:= '192.168.10.10.4.1', 
	nSlaveAddr:=1041,   //模切缓存
	nSubIndex:=0 , 
	nIndex:=16#2108 ,   //  平滑时间
	pSrcBuf:=ADR(SEPTATCache_fSmoothValue[3]),       //写入参数值 
	cbBufLen:=SIZEOF(SEPTATCache_fSmoothValue[3]),    
	bExecute:= SEPTATCache_bWriteCoeValue[3],    
	tTimeout:= T#3S, 
	bBusy=> , 
	bError=> , 
	nErrId=> );
//保存	
FB_EcCoESdoWrite_CaSEPTATCache[3](
	sNetId:= '192.168.10.10.4.1', 
	nSlaveAddr:=1041 ,   //模切缓存
	nSubIndex:=0 , 
	nIndex:=16#2108 ,   // 平滑时间
	pSrcBuf:=ADR(wSaveCoeCode),      //保存参数值
	cbBufLen:=SIZEOF(wSaveCoeCode),    
	bExecute:= SEPTATCache_SavePara[3],    
	tTimeout:= T#3S, 
	bBusy=> , 
	bError=> , 
	nErrId=> );	
	
	
	
	
	
//写入	
FB_EcCoESdoWrite_CaSEPTATCache[2](
	sNetId:='192.168.10.10.4.1', 
	nSlaveAddr:=1041 ,   //模切缓存
	nSubIndex:=0 , 
	nIndex:=16#2109 ,   // 平滑方式
	pSrcBuf:=ADR(SEPTATCache_fSmoothValue[4]),       //写入参数值 
	cbBufLen:=SIZEOF(SEPTATCache_fSmoothValue[4]),    
	bExecute:= SEPTATCache_bWriteCoeValue[4],    
	tTimeout:= T#3S, 
	bBusy=> , 
	bError=> , 
	nErrId=> );
//保存	
FB_EcCoESdoWrite_CaSEPTATCache[4](
	sNetId:= '192.168.10.10.4.1', 
	nSlaveAddr:=1041,   //模切缓存
	nSubIndex:=0 , 
	nIndex:=16#2109 ,   // 平滑方式
	pSrcBuf:=ADR(wSaveCoeCode),      //保存参数值
	cbBufLen:=SIZEOF(wSaveCoeCode),    
	bExecute:= SEPTATCache_SavePara[4],    
	tTimeout:= T#3S, 
	bBusy=> , 
	bError=> , 
	nErrId=> );	


	
	
	
	

//负极模切主驱\
//写入
FB_EcCoESdoWrite_CaDriverDDR[1](
	sNetId:= '192.168.10.10.4.1', 
	nSlaveAddr:=1042 ,   //模切主驱
	nSubIndex:=0 , 
	nIndex:=16#2108 ,   //  平滑时间
	pSrcBuf:=ADR(DriverDDR_fSmoothValue[3]),       //写入参数值 
	cbBufLen:=SIZEOF(DriverDDR_fSmoothValue[3]),    
	bExecute:= DriverDDR_bWriteCoeValue[3],    
	tTimeout:= T#3S, 
	bBusy=> , 
	bError=> , 
	nErrId=> );
//保存	
FB_EcCoESdoWrite_CaDriverDDR[3](
	sNetId:= '192.168.10.10.4.1', 
	nSlaveAddr:=1042 ,   //模切主驱
	nSubIndex:=0 , 
	nIndex:=16#2108 ,   // 平滑时间
	pSrcBuf:=ADR(wSaveCoeCode),      //保存参数值
	cbBufLen:=SIZEOF(wSaveCoeCode),    
	bExecute:= DriverDDR_SavePara[3],    
	tTimeout:= T#3S, 
	bBusy=> , 
	bError=> , 
	nErrId=> );	
	
	
	
	
	
//写入	
FB_EcCoESdoWrite_CaDriverDDR[2](
	sNetId:='192.168.10.10.4.1', 
	nSlaveAddr:=1042 ,   //模切主驱
	nSubIndex:=0 , 
	nIndex:=16#2109 ,   // 平滑方式
	pSrcBuf:=ADR(DriverDDR_fSmoothValue[4]),       //写入参数值 
	cbBufLen:=SIZEOF(DriverDDR_fSmoothValue[4]),    
	bExecute:= DriverDDR_bWriteCoeValue[4],    
	tTimeout:= T#3S, 
	bBusy=> , 
	bError=> , 
	nErrId=> );	
//保存	
FB_EcCoESdoWrite_CaDriverDDR[4](
	sNetId:= '192.168.10.10.4.1', 
	nSlaveAddr:=1042 ,   //模切主驱
	nSubIndex:=0 , 
	nIndex:=16#2109 ,   // 平滑方式
	pSrcBuf:=ADR(wSaveCoeCode),      //保存参数值
	cbBufLen:=SIZEOF(wSaveCoeCode),    
	bExecute:= DriverDDR_SavePara[4],    
	tTimeout:= T#3S, 
	bBusy=> , 
	bError=> , 
	nErrId=> );	
	
	
	*)
END_ACTION

ACTION MotionBasic:


//
FOR i:=1 TO MaxAxes DO
IF i<>9 AND i<>33 AND i<>20 AND i<>21 AND i<>22 AND i<>44 AND i<>45 AND i<>46   THEN
  	arrAxisCtrl[i].Cmd.JogN_Condition:=NOT arrAxisCtrl[i].Io.biNegLimit;
	arrAxisCtrl[i].Cmd.JogP_Condition:=NOT arrAxisCtrl[i].Io.biPosLimit;
END_IF		
	csAxis[i](bReset:=stSysState.bReset , Axis:=arrAxis[i] , stAxisCtrl:=arrAxisCtrl[i] , stAxisPar:=arrAxisPar[i] );
	arrAxisPar[i].fHomeSlowSpeed:=arrAxisPar[i].fHomeFastSpeed/5;
END_FOR

FOR i:=1 TO MaxDust DO
  fbDustMotor[i](stSetpMotor:=arrDustMotor[i]);
END_FOR

FOR i:=1 TO NumOfDrives DO
  arrAxisCtrl[i].Status.bDrivesOP:=DrivesOP[i]=8;//(DrivesOP[i]=8 AND i<>3 AND i<>27) OR (DrivesOP[i]=10 AND (i=3 OR i=27));
END_FOR

fbAnSetp1Moter(stSetpMotor:=AnSetpMotor );//正极NG排杆电机
fbCaSetp1Moter(stSetpMotor:=CaSetpMotor );//负极NG排杆电机

IF ABS(iTargetTorque[1])>150 THEN
	iTargetTorque[1]:=0;
END_IF
IF ABS(iTargetTorque[2])>150 THEN
	iTargetTorque[2]:=0;
END_IF

//////////////张力摆杆超速后断开使能////////
IF (arrAxisCtrl[NameNo.AnAxisNo.PoleTension].Io.biNegLimit OR arrAxisCtrl[NameNo.AnAxisNo.PoleTension].Io.biPosLimit) AND arrAxisCtrl[NameNo.AnAxisNo.PoleTension].Status.fActVelo>500 THEN
	arrAxisCtrl[NameNo.AnAxisNo.PoleTension].Cmd.bEnable:=FALSE;
END_IF
IF (arrAxisCtrl[NameNo.CaAxisNo.PoleTension].Io.biNegLimit OR arrAxisCtrl[NameNo.CaAxisNo.PoleTension].Io.biPosLimit) AND arrAxisCtrl[NameNo.CaAxisNo.PoleTension].Status.fActVelo>500 THEN
	arrAxisCtrl[NameNo.CaAxisNo.PoleTension].Cmd.bEnable:=FALSE;
END_IF

//////////主轴参数放大////////
arrAxisPar[NameNo.AnVirAxisNo.VirMain].fMaxVel:=8000;
arrAxisPar[NameNo.AnVirAxisNo.VirMain].fMaxAccDec:=300000;
arrAxisPar[NameNo.AnVirAxisNo.VirMain].fConVelPercentage:=0.8;
arrAxisPar[NameNo.CaVirAxisNo.VirMain].fMaxVel:=8000;
arrAxisPar[NameNo.CaVirAxisNo.VirMain].fMaxAccDec:=300000;
arrAxisPar[NameNo.CaVirAxisNo.VirMain].fConVelPercentage:=0.8;
END_ACTION

ACTION MS_Alarm:
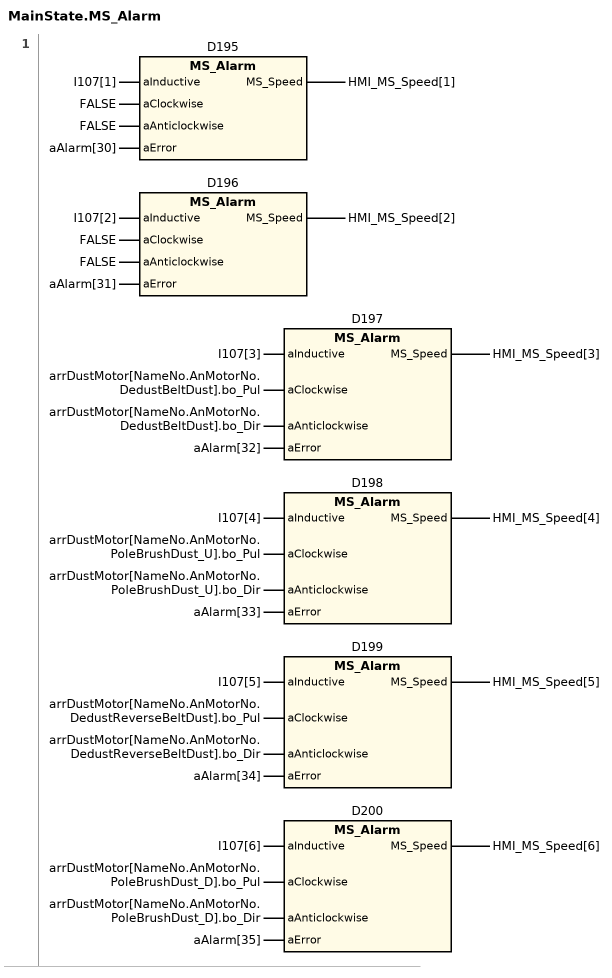
// NETWORK 1
D195(aInductive := I107[1], aClockwise := FALSE, aAnticlockwise := FALSE, aError := aAlarm[30]); // MS_Alarm
HMI_MS_Speed[1] := D195.MS_Speed;
D196(aInductive := I107[2], aClockwise := FALSE, aAnticlockwise := FALSE, aError := aAlarm[31]); // MS_Alarm
HMI_MS_Speed[2] := D196.MS_Speed;
D197(
    aInductive := I107[3],
    aClockwise := arrDustMotor[NameNo.AnMotorNo.DedustBeltDust].bo_Pul,
    aAnticlockwise := arrDustMotor[NameNo.AnMotorNo.DedustBeltDust].bo_Dir,
    aError := aAlarm[32]); // MS_Alarm
HMI_MS_Speed[3] := D197.MS_Speed;
D198(
    aInductive := I107[4],
    aClockwise := arrDustMotor[NameNo.AnMotorNo.PoleBrushDust_U].bo_Pul,
    aAnticlockwise := arrDustMotor[NameNo.AnMotorNo.PoleBrushDust_U].bo_Dir,
    aError := aAlarm[33]); // MS_Alarm
HMI_MS_Speed[4] := D198.MS_Speed;
D199(
    aInductive := I107[5],
    aClockwise := arrDustMotor[NameNo.AnMotorNo.DedustReverseBeltDust].bo_Pul,
    aAnticlockwise := arrDustMotor[NameNo.AnMotorNo.DedustReverseBeltDust].bo_Dir,
    aError := aAlarm[34]); // MS_Alarm
HMI_MS_Speed[5] := D199.MS_Speed;
D200(
    aInductive := I107[6],
    aClockwise := arrDustMotor[NameNo.AnMotorNo.PoleBrushDust_D].bo_Pul,
    aAnticlockwise := arrDustMotor[NameNo.AnMotorNo.PoleBrushDust_D].bo_Dir,
    aError := aAlarm[35]); // MS_Alarm
HMI_MS_Speed[6] := D200.MS_Speed;

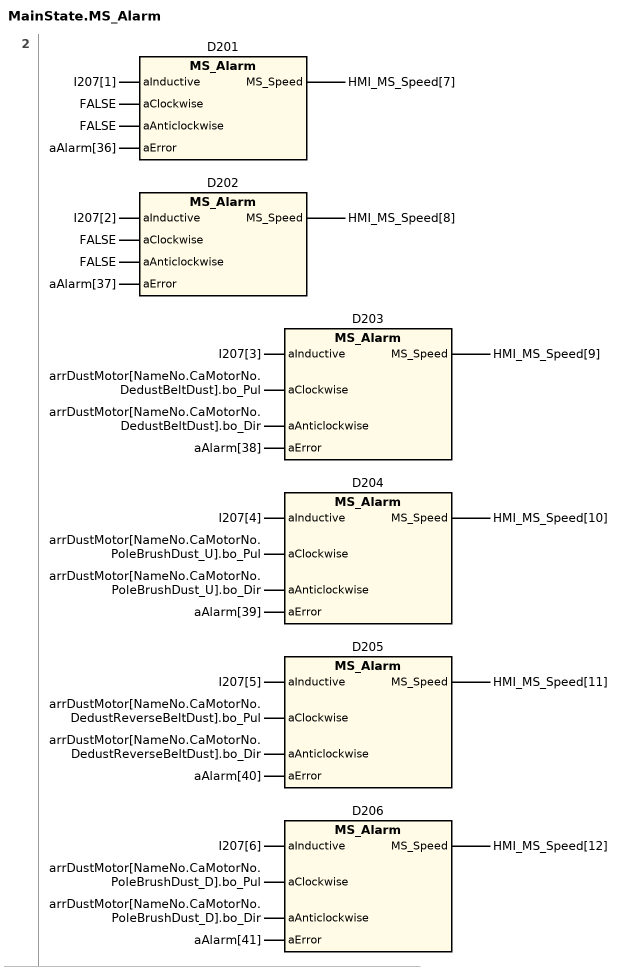
// NETWORK 2
D201(aInductive := I207[1], aClockwise := FALSE, aAnticlockwise := FALSE, aError := aAlarm[36]); // MS_Alarm
HMI_MS_Speed[7] := D201.MS_Speed;
D202(aInductive := I207[2], aClockwise := FALSE, aAnticlockwise := FALSE, aError := aAlarm[37]); // MS_Alarm
HMI_MS_Speed[8] := D202.MS_Speed;
D203(
    aInductive := I207[3],
    aClockwise := arrDustMotor[NameNo.CaMotorNo.DedustBeltDust].bo_Pul,
    aAnticlockwise := arrDustMotor[NameNo.CaMotorNo.DedustBeltDust].bo_Dir,
    aError := aAlarm[38]); // MS_Alarm
HMI_MS_Speed[9] := D203.MS_Speed;
D204(
    aInductive := I207[4],
    aClockwise := arrDustMotor[NameNo.CaMotorNo.PoleBrushDust_U].bo_Pul,
    aAnticlockwise := arrDustMotor[NameNo.CaMotorNo.PoleBrushDust_U].bo_Dir,
    aError := aAlarm[39]); // MS_Alarm
HMI_MS_Speed[10] := D204.MS_Speed;
D205(
    aInductive := I207[5],
    aClockwise := arrDustMotor[NameNo.CaMotorNo.DedustReverseBeltDust].bo_Pul,
    aAnticlockwise := arrDustMotor[NameNo.CaMotorNo.DedustReverseBeltDust].bo_Dir,
    aError := aAlarm[40]); // MS_Alarm
HMI_MS_Speed[11] := D205.MS_Speed;
D206(
    aInductive := I207[6],
    aClockwise := arrDustMotor[NameNo.CaMotorNo.PoleBrushDust_D].bo_Pul,
    aAnticlockwise := arrDustMotor[NameNo.CaMotorNo.PoleBrushDust_D].bo_Dir,
    aError := aAlarm[41]); // MS_Alarm
HMI_MS_Speed[12] := D206.MS_Speed;

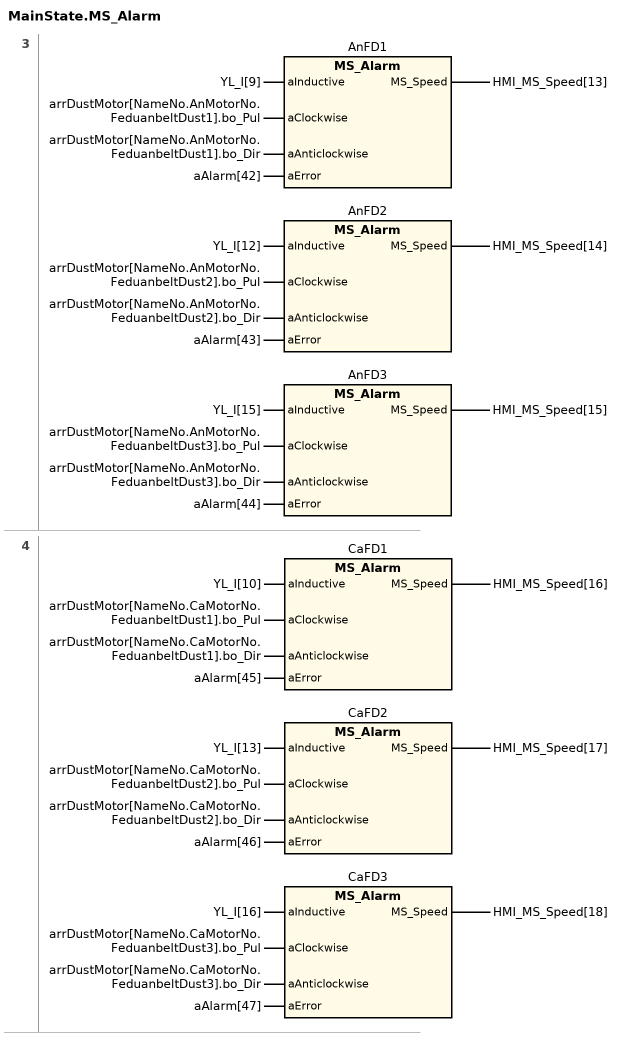
// NETWORK 3
AnFD1(
    aInductive := YL_I[9],
    aClockwise := arrDustMotor[NameNo.AnMotorNo.FeduanbeltDust1].bo_Pul,
    aAnticlockwise := arrDustMotor[NameNo.AnMotorNo.FeduanbeltDust1].bo_Dir,
    aError := aAlarm[42]); // MS_Alarm
HMI_MS_Speed[13] := AnFD1.MS_Speed;
AnFD2(
    aInductive := YL_I[12],
    aClockwise := arrDustMotor[NameNo.AnMotorNo.FeduanbeltDust2].bo_Pul,
    aAnticlockwise := arrDustMotor[NameNo.AnMotorNo.FeduanbeltDust2].bo_Dir,
    aError := aAlarm[43]); // MS_Alarm
HMI_MS_Speed[14] := AnFD2.MS_Speed;
AnFD3(
    aInductive := YL_I[15],
    aClockwise := arrDustMotor[NameNo.AnMotorNo.FeduanbeltDust3].bo_Pul,
    aAnticlockwise := arrDustMotor[NameNo.AnMotorNo.FeduanbeltDust3].bo_Dir,
    aError := aAlarm[44]); // MS_Alarm
HMI_MS_Speed[15] := AnFD3.MS_Speed;

// NETWORK 4
CaFD1(
    aInductive := YL_I[10],
    aClockwise := arrDustMotor[NameNo.CaMotorNo.FeduanbeltDust1].bo_Pul,
    aAnticlockwise := arrDustMotor[NameNo.CaMotorNo.FeduanbeltDust1].bo_Dir,
    aError := aAlarm[45]); // MS_Alarm
HMI_MS_Speed[16] := CaFD1.MS_Speed;
CaFD2(
    aInductive := YL_I[13],
    aClockwise := arrDustMotor[NameNo.CaMotorNo.FeduanbeltDust2].bo_Pul,
    aAnticlockwise := arrDustMotor[NameNo.CaMotorNo.FeduanbeltDust2].bo_Dir,
    aError := aAlarm[46]); // MS_Alarm
HMI_MS_Speed[17] := CaFD2.MS_Speed;
CaFD3(
    aInductive := YL_I[16],
    aClockwise := arrDustMotor[NameNo.CaMotorNo.FeduanbeltDust3].bo_Pul,
    aAnticlockwise := arrDustMotor[NameNo.CaMotorNo.FeduanbeltDust3].bo_Dir,
    aError := aAlarm[47]); // MS_Alarm
HMI_MS_Speed[18] := CaFD3.MS_Speed;
END_ACTION

ACTION Pusle:

/////////////////////////////////////////时钟脉冲////////////////////////////////////////////////////////////
//fbPulseCtrl1(PT_OFF:=T#2MS, PT_ON:=T#2MS, Q=>, RT=>);
fbPulseCtrl[1](PT_OFF:=T#2MS, PT_ON:=T#2MS,   );
fbPulseCtrl[2](PT_OFF:=T#4MS, PT_ON:=T#4MS,    );
fbPulseCtrl[3](PT_OFF:=T#10MS, PT_ON:=T#10MS,   );

fbPulseCtrl[4](PT_OFF:=T#50MS, PT_ON:=T#50MS,   );
fbPulseCtrl[5](PT_OFF:=T#3S, PT_ON:=T#3S,    );
fbPulseCtrl[6](PT_OFF:=T#5S, PT_ON:=T#5S,   );

fbPulseCtrl[8](PT_OFF:=T#250MS, PT_ON:=T#250MS,   );

fbPulseCtrl[9](PT_OFF:=T#2S, PT_ON:=T#200MS,   );
fbPulseCtrl[10](PT_OFF:=T#10S, PT_ON:=T#10S,   );
fbPulseCtrl[1].Q;
fbPulseCtrl[1].RT;
fbPulseCtrl[2].Q;
fbPulseCtrl[2].RT;
fbPulseCtrl[3].Q;
fbPulseCtrl[3].RT;
fbPulseCtrl[4].Q;
fbPulseCtrl[4].RT;
fbPulseCtrl[5].Q;
fbPulseCtrl[5].RT;
fbPulseCtrl[6].Q;
fbPulseCtrl[6].RT;

fbPulseCtrl[8].Q;
fbPulseCtrl[8].RT;
fbPulseCtrl[9].Q;
fbPulseCtrl[9].RT;
fbPulseCtrl[10].Q;
fbPulseCtrl[10].RT;
(*
IF bWaterOn AND ( bWaterOn2   OR    ABS( arrAxisCtrl[P1AxisNo.GMWind_U].Status.fActVelo)>=5 AND  ABS (arrAxisCtrl[P1AxisNo.GMWind_D].Status.fActVelo)>=5 )   THEN
  //P3EL2889S[3,5]:= fbPulseCtrl[9].Q;
   P1EL2889S[3,1]:= fbPulseCtrl[9].Q;
   P1EL2889S[3,2]:= fbPulseCtrl[9].Q;

   P2EL2889S[4,1]:=fbPulseCtrl[9].Q	;	
   P2EL2889S[4,2]:=fbPulseCtrl[9].Q;	

   P2EL2889S[4,3]:=fbPulseCtrl[9].Q	;	
   P2EL2889S[4,4]:=fbPulseCtrl[9].Q;	

ELSE
  //P3EL2889S[3,5]:= FALSE;
   P1EL2889S[3,1]:= FALSE;
   P1EL2889S[3,2]:= FALSE;
   P2EL2889S[4,1]:= FALSE	;	
   P2EL2889S[4,2]:= FALSE;	

   P2EL2889S[4,3]:=FALSE	;	
   P2EL2889S[4,4]:=FALSE;	
END_IF


//P1EL2889S[3,1]

*)
END_ACTION

ACTION RecBasic:
//纠偏控制
FOR i:=1 TO MaxRec DO
    fbRec[i]( RecCtrl:=arrRecCtrl[i] );
END_FOR
END_ACTION

END_PROGRAM

(* stored: Version 1.1.0.1, ProductVersion 3.1.4024.12
   POU MainState: Id {6ef34fba-d1da-4e27-9ef0-ec34a9427286}, SpecialFunc None
   Action Alarm: Id {4b075792-06ef-4c2e-843f-ecf9e6644509}
   Action Condition: Id {f7c3c673-ccf9-4740-950e-c5d8fbe37c32}
   Action CyBasic: Id {d7ad8c6c-fc6e-4e69-870d-5eea8b8486ad}
   Action EStop: Id {b7a6d35a-ed44-46ea-a2dd-d41fc75526df}
   Action Init: Id {633e6e37-7817-421e-8123-21afc873bea3}
   Action MesCollect: Id {6bd430c5-ec81-43cd-9ebc-4ae4a6278f2c}
   Action Motion_coe: Id {576cd356-9582-442a-bbbc-8efa32d5392c}
   Action MotionBasic: Id {3a0b1861-7a08-44c7-b364-48f37a0928ea}
   Action MS_Alarm: Id {4634da08-ba6a-4762-bdfb-a0841f3476df}
   Action Pusle: Id {ed1aaec7-93f9-45d4-9266-e4f9208b4061}
   Action RecBasic: Id {e63bc7b7-ea9e-475f-ad46-8a86744fc463} *)
